LIN {X 0.035,Y -624.927,Z 1269.319,A 0.000,B 0.000,C 90.000,E1 93.326} C_DIS
LIN {X 0.207,Y -616.621,Z 1269.315,A 0.000,B 0.000,C 90.000,E1 92.636} C_DIS
LIN {X -0.076,Y -609.408,Z 1269.312,A 0.000,B 0.000,C 90.000,E1 92.121} C_DIS
LIN {X -0.106,Y -601.874,Z 1269.309,A 0.000,B 0.000,C 90.000,E1 91.604} C_DIS
LIN {X 0.134,Y -595.870,Z 1269.307,A 0.000,B 0.000,C 90.000,E1 91.203} C_DIS
LIN {X -0.159,Y -588.937,Z 1269.305,A 0.000,B 0.000,C 90.000,E1 90.859} C_DIS
LIN {X 0.273,Y -583.448,Z 1269.303,A 0.000,B 0.000,C 90.000,E1 90.573} C_DIS
LIN {X -0.248,Y -576.328,Z 1269.302,A 0.000,B 0.000,C 90.000,E1 90.344} C_DIS
LIN {X -0.083,Y -571.719,Z 1269.301,A 0.000,B 0.000,C 90.000,E1 90.115} C_DIS
LIN {X -0.130,Y -571.653,Z 1269.301,A 0.000,B 0.000,C 90.000,E1 90.115} C_DIS
LIN {X -0.005,Y -570.486,Z 1269.300,A 0.000,B 0.000,C 90.000,E1 89.943} C_DIS
LIN {X -0.259,Y -568.764,Z 1269.299,A 0.000,B 0.000,C 90.000,E1 89.771} C_DIS
LIN {X 0.268,Y -568.741,Z 1269.299,A 0.000,B 0.000,C 90.000,E1 89.714} C_DIS
LIN {X 0.075,Y -568.279,Z 1269.297,A 0.000,B 0.000,C 90.000,E1 89.370} C_DIS
LIN {X 0.099,Y -568.544,Z 1269.293,A 0.000,B 0.000,C 90.000,E1 88.682} C_DIS
LIN {X 0.005,Y -570.330,Z 1269.281,A 0.000,B 0.000,C 90.000,E1 86.502} C_DIS
LIN {X -0.257,Y -573.067,Z 1269.266,A 0.000,B 0.000,C 90.000,E1 83.799} C_DIS
LIN {X -0.006,Y -574.512,Z 1269.258,A 0.000,B 0.000,C 90.000,E1 82.413} C_DIS
LIN {X 0.063,Y -575.760,Z 1269.252,A 0.000,B 0.000,C 90.000,E1 81.319} C_DIS
LIN {X -0.129,Y -577.174,Z 1269.244,A 0.000,B 0.000,C 90.000,E1 79.982} C_DIS
LIN {X 0.162,Y -578.183,Z 1269.238,A 0.000,B 0.000,C 90.000,E1 78.870} C_DIS
LIN {X -0.213,Y -579.536,Z 1269.229,A 0.000,B 0.000,C 90.000,E1 77.285} C_DIS
LIN {X 0.115,Y -580.341,Z 1269.223,A 0.000,B 0.000,C 90.000,E1 76.172} C_DIS
LIN {X -0.086,Y -581.484,Z 1269.214,A 0.000,B 0.000,C 90.000,E1 74.574} C_DIS
LIN {X 0.110,Y -582.570,Z 1269.204,A 0.000,B 0.000,C 90.000,E1 72.670} C_DIS
LIN {X 0.220,Y -583.261,Z 1269.198,A 0.000,B 0.000,C 90.000,E1 71.583} C_DIS
LIN {X -0.147,Y -584.186,Z 1269.189,A 0.000,B 0.000,C 90.000,E1 70.007} C_DIS
LIN {X -0.142,Y -585.613,Z 1269.176,A 0.000,B 0.000,C 90.000,E1 67.592} C_DIS
LIN {X 0.272,Y -587.301,Z 1269.164,A 0.000,B 0.000,C 90.000,E1 65.409} C_DIS
LIN {X -0.020,Y -588.370,Z 1269.156,A 0.000,B 0.000,C 90.000,E1 64.101} C_DIS
LIN {X -0.109,Y -590.186,Z 1269.144,A 0.000,B 0.000,C 90.000,E1 61.975} C_DIS
LIN {X -0.172,Y -591.757,Z 1269.135,A 0.000,B 0.000,C 90.000,E1 60.383} C_DIS
LIN {X -0.394,Y -593.165,Z 1269.128,A 0.000,B 0.000,C 90.000,E1 59.076} C_DIS
LIN {X 0.019,Y -594.578,Z 1269.121,A 0.000,B 0.000,C 90.000,E1 57.709} C_DIS
LIN {X -0.137,Y -596.161,Z 1269.112,A 0.000,B 0.000,C 90.000,E1 56.135} C_DIS
LIN {X 0.075,Y -597.715,Z 1269.103,A 0.000,B 0.000,C 90.000,E1 54.529} C_DIS
LIN {X -0.172,Y -599.043,Z 1269.094,A 0.000,B 0.000,C 90.000,E1 52.970} C_DIS
LIN {X -0.032,Y -600.276,Z 1269.085,A 0.000,B 0.000,C 90.000,E1 51.376} C_DIS
LIN {X -0.367,Y -601.098,Z 1269.080,A 0.000,B 0.000,C 90.000,E1 50.356} C_DIS
LIN {X -0.097,Y -601.474,Z 1269.075,A 0.000,B 0.000,C 90.000,E1 49.542} C_DIS
LIN {X -0.018,Y -602.330,Z 1269.064,A 0.000,B 0.000,C 90.000,E1 47.433} C_DIS
LIN {X -0.156,Y -602.728,Z 1269.056,A 0.000,B 0.000,C 90.000,E1 46.134} C_DIS
LIN {X 0.091,Y -602.846,Z 1269.052,A 0.000,B 0.000,C 90.000,E1 45.324} C_DIS
LIN {X -0.063,Y -602.734,Z 1269.045,A 0.000,B 0.000,C 90.000,E1 44.028} C_DIS
LIN {X -0.024,Y -602.493,Z 1269.039,A 0.000,B 0.000,C 90.000,E1 42.975} C_DIS
LIN {X 0.077,Y -601.909,Z 1269.030,A 0.000,B 0.000,C 90.000,E1 41.391} C_DIS
LIN {X 0.179,Y -601.206,Z 1269.021,A 0.000,B 0.000,C 90.000,E1 39.806} C_DIS
LIN {X 0.231,Y -600.557,Z 1269.016,A 0.000,B 0.000,C 90.000,E1 38.749} C_DIS
LIN {X -0.104,Y -599.810,Z 1269.010,A 0.000,B 0.000,C 90.000,E1 37.729} C_DIS
LIN {X 0.267,Y -598.410,Z 1269.002,A 0.000,B 0.000,C 90.000,E1 36.377} C_DIS
LIN {X -0.218,Y -596.615,Z 1268.995,A 0.000,B 0.000,C 90.000,E1 35.105} C_DIS
LIN {X -0.248,Y -594.236,Z 1268.988,A 0.000,B 0.000,C 90.000,E1 33.785} C_DIS
LIN {X 0.075,Y -592.556,Z 1268.983,A 0.000,B 0.000,C 90.000,E1 32.959} C_DIS
LIN {X 0.173,Y -591.315,Z 1268.980,A 0.000,B 0.000,C 90.000,E1 32.418} C_DIS
LIN {X -0.160,Y -588.416,Z 1268.974,A 0.000,B 0.000,C 90.000,E1 31.386} C_DIS
LIN {X -0.215,Y -585.793,Z 1268.970,A 0.000,B 0.000,C 90.000,E1 30.590} C_DIS
LIN {X -0.167,Y -583.891,Z 1268.967,A 0.000,B 0.000,C 90.000,E1 30.050} C_DIS
LIN {X 0.238,Y -580.550,Z 1268.962,A 0.000,B 0.000,C 90.000,E1 29.205} C_DIS
LIN {X 0.026,Y -576.284,Z 1268.957,A 0.000,B 0.000,C 90.000,E1 28.281} C_DIS
LIN {X 0.075,Y -571.866,Z 1268.953,A 0.000,B 0.000,C 90.000,E1 27.462} C_DIS
LIN {X -0.166,Y -567.213,Z 1268.948,A 0.000,B 0.000,C 90.000,E1 26.668} C_DIS
LIN {X -0.204,Y -561.915,Z 1268.943,A 0.000,B 0.000,C 90.000,E1 25.848} C_DIS
LIN {X -0.191,Y -557.238,Z 1268.940,A 0.000,B 0.000,C 90.000,E1 25.155} C_DIS
LIN {X -0.002,Y -554.199,Z 1268.937,A 0.000,B 0.000,C 90.000,E1 24.719} C_DIS
LIN {X -0.172,Y -547.673,Z 1268.933,A 0.000,B 0.000,C 90.000,E1 23.898} C_DIS
LIN {X 0.087,Y -540.497,Z 1268.928,A 0.000,B 0.000,C 90.000,E1 23.025} C_DIS
LIN {X 0.186,Y -536.683,Z 1268.926,A 0.000,B 0.000,C 90.000,E1 22.589} C_DIS
LIN {X -0.022,Y -527.764,Z 1268.920,A 0.000,B 0.000,C 90.000,E1 21.642} C_DIS
LIN {X 0.012,Y -518.433,Z 1268.915,A 0.000,B 0.000,C 90.000,E1 20.663} C_DIS
LIN {X -0.089,Y -507.507,Z 1268.909,A 0.000,B 0.000,C 90.000,E1 19.577} C_DIS
LIN {X 0.166,Y -497.766,Z 1268.903,A 0.000,B 0.000,C 90.000,E1 18.598} C_DIS
LIN {X -0.088,Y -489.206,Z 1268.899,A 0.000,B 0.000,C 90.000,E1 17.819} C_DIS
LIN {X -0.222,Y -480.567,Z 1268.895,A 0.000,B 0.000,C 90.000,E1 17.040} C_DIS
LIN {X -0.066,Y -467.187,Z 1268.888,A 0.000,B 0.000,C 90.000,E1 15.843} C_DIS
LIN {X 0.059,Y -446.488,Z 1268.878,A 0.000,B 0.000,C 90.000,E1 13.939} C_DIS
LIN {X -0.007,Y -429.004,Z 1268.868,A 0.000,B 0.000,C 90.000,E1 12.243} C_DIS
LIN {X -0.023,Y -411.922,Z 1268.858,A 0.000,B 0.000,C 90.000,E1 10.433} C_DIS
LIN {X 0.080,Y -402.151,Z 1268.852,A 0.000,B 0.000,C 90.000,E1 9.321} C_DIS
LIN {X -0.078,Y -398.253,Z 1268.849,A 0.000,B 0.000,C 90.000,E1 8.859} C_DIS
LIN {X 0.174,Y -395.068,Z 1268.847,A 0.000,B 0.000,C 90.000,E1 8.341} C_DIS
LIN {X 0.205,Y -394.907,Z 1268.846,A 0.000,B 0.000,C 90.000,E1 8.276} C_DIS
LIN {X 0.167,Y -394.904,Z 1268.846,A 0.000,B 0.000,C 90.000,E1 8.276} C_DIS
LIN {X -0.182,Y -395.576,Z 1268.845,A 0.000,B 0.000,C 90.000,E1 8.106} C_DIS
LIN {X -0.008,Y -396.125,Z 1268.844,A 0.000,B 0.000,C 90.000,E1 7.992} C_DIS
LIN {X 0.069,Y -399.536,Z 1268.843,A 0.000,B 0.000,C 90.000,E1 7.644} C_DIS
LIN {X -0.190,Y -401.491,Z 1268.842,A 0.000,B 0.000,C 90.000,E1 7.530} C_DIS
LIN {X -0.044,Y -408.684,Z 1268.839,A 0.000,B 0.000,C 90.000,E1 7.068} C_DIS
LIN {X -0.067,Y -413.477,Z 1268.838,A 0.000,B 0.000,C 90.000,E1 6.777} C_DIS
LIN {X 0.129,Y -419.785,Z 1268.835,A 0.000,B 0.000,C 90.000,E1 6.315} C_DIS
LIN {X 0.092,Y -426.124,Z 1268.833,A 0.000,B 0.000,C 90.000,E1 5.853} C_DIS
LIN {X 0.180,Y -435.617,Z 1268.828,A 0.000,B 0.000,C 90.000,E1 5.106} C_DIS
LIN {X -0.122,Y -443.387,Z 1268.825,A 0.000,B 0.000,C 90.000,E1 4.531} C_DIS
LIN {X 0.118,Y -454.124,Z 1268.820,A 0.000,B 0.000,C 90.000,E1 3.612} C_DIS
LIN {X -0.027,Y -461.487,Z 1268.817,A 0.000,B 0.000,C 90.000,E1 2.980} C_DIS
LIN {X -0.200,Y -467.315,Z 1268.814,A 0.000,B 0.000,C 90.000,E1 2.465} C_DIS
LIN {X 0.179,Y -474.204,Z 1268.810,A 0.000,B 0.000,C 90.000,E1 1.718} C_DIS
LIN {X 0.163,Y -479.557,Z 1268.807,A 0.000,B 0.000,C 90.000,E1 1.146} C_DIS
LIN {X -0.200,Y -487.318,Z 1268.802,A 0.000,B 0.000,C 90.000,E1 0.286} C_DIS
LIN {X 0.026,Y -493.312,Z 1268.797,A 0.000,B 0.000,C 90.000,E1 359.484} C_DIS
LIN {X -0.091,Y -498.725,Z 1268.793,A 0.000,B 0.000,C 90.000,E1 358.740} C_DIS
LIN {X 0.049,Y -504.636,Z 1268.788,A 0.000,B 0.000,C 90.000,E1 357.822} C_DIS
LIN {X -0.171,Y -508.377,Z 1268.785,A 0.000,B 0.000,C 90.000,E1 357.249} C_DIS
LIN {X -0.132,Y -512.702,Z 1268.781,A 0.000,B 0.000,C 90.000,E1 356.502} C_DIS
LIN {X 0.249,Y -516.047,Z 1268.777,A 0.000,B 0.000,C 90.000,E1 355.869} C_DIS
LIN {X -0.149,Y -519.875,Z 1268.773,A 0.000,B 0.000,C 90.000,E1 355.179} C_DIS
LIN {X 0.003,Y -523.393,Z 1268.769,A 0.000,B 0.000,C 90.000,E1 354.432} C_DIS
LIN {X 0.199,Y -527.979,Z 1268.763,A 0.000,B 0.000,C 90.000,E1 353.394} C_DIS
LIN {X -0.078,Y -531.971,Z 1268.758,A 0.000,B 0.000,C 90.000,E1 352.413} C_DIS
LIN {X -0.036,Y -535.135,Z 1268.753,A 0.000,B 0.000,C 90.000,E1 351.546} C_DIS
LIN {X 0.039,Y -537.984,Z 1268.748,A 0.000,B 0.000,C 90.000,E1 350.679} C_DIS
LIN {X 0.233,Y -540.592,Z 1268.744,A 0.000,B 0.000,C 90.000,E1 349.803} C_DIS
LIN {X -0.094,Y -543.724,Z 1268.737,A 0.000,B 0.000,C 90.000,E1 348.701} C_DIS
LIN {X 0.075,Y -545.161,Z 1268.734,A 0.000,B 0.000,C 90.000,E1 348.117} C_DIS
LIN {X 0.130,Y -548.295,Z 1268.726,A 0.000,B 0.000,C 90.000,E1 346.700} C_DIS
LIN {X -0.098,Y -549.960,Z 1268.722,A 0.000,B 0.000,C 90.000,E1 345.880} C_DIS
LIN {X -0.067,Y -551.925,Z 1268.715,A 0.000,B 0.000,C 90.000,E1 344.755} C_DIS
LIN {X 0.144,Y -553.533,Z 1268.709,A 0.000,B 0.000,C 90.000,E1 343.614} C_DIS
LIN {X 0.110,Y -554.552,Z 1268.704,A 0.000,B 0.000,C 90.000,E1 342.779} C_DIS
LIN {X -0.164,Y -555.602,Z 1268.698,A 0.000,B 0.000,C 90.000,E1 341.692} C_DIS
LIN {X -0.187,Y -556.065,Z 1268.694,A 0.000,B 0.000,C 90.000,E1 340.859} C_DIS
LIN {X -0.131,Y -556.226,Z 1268.691,A 0.000,B 0.000,C 90.000,E1 340.296} C_DIS
LIN {X 0.035,Y -556.128,Z 1268.686,A 0.000,B 0.000,C 90.000,E1 339.444} C_DIS
LIN {X 0.195,Y -555.751,Z 1268.681,A 0.000,B 0.000,C 90.000,E1 338.592} C_DIS
LIN {X 0.119,Y -554.781,Z 1268.675,A 0.000,B 0.000,C 90.000,E1 337.486} C_DIS
LIN {X -0.042,Y -553.574,Z 1268.670,A 0.000,B 0.000,C 90.000,E1 336.666} C_DIS
LIN {X 0.294,Y -552.191,Z 1268.666,A 0.000,B 0.000,C 90.000,E1 335.793} C_DIS
LIN {X 0.144,Y -549.562,Z 1268.658,A 0.000,B 0.000,C 90.000,E1 334.409} C_DIS
LIN {X 0.167,Y -547.974,Z 1268.655,A 0.000,B 0.000,C 90.000,E1 333.845} C_DIS
LIN {X -0.072,Y -547.336,Z 1268.653,A 0.000,B 0.000,C 90.000,E1 333.589} C_DIS
LIN {X -0.066,Y -544.751,Z 1268.649,A 0.000,B 0.000,C 90.000,E1 332.743} C_DIS
LIN {X 0.170,Y -542.787,Z 1268.645,A 0.000,B 0.000,C 90.000,E1 332.153} C_DIS
LIN {X 0.000,Y -538.988,Z 1268.640,A 0.000,B 0.000,C 90.000,E1 331.179} C_DIS
LIN {X -0.086,Y -534.890,Z 1268.635,A 0.000,B 0.000,C 90.000,E1 330.333} C_DIS
LIN {X -0.074,Y -530.995,Z 1268.631,A 0.000,B 0.000,C 90.000,E1 329.616} C_DIS
LIN {X 0.169,Y -526.763,Z 1268.627,A 0.000,B 0.000,C 90.000,E1 328.869} C_DIS
LIN {X -0.179,Y -517.818,Z 1268.619,A 0.000,B 0.000,C 90.000,E1 327.454} C_DIS
LIN {X -0.054,Y -513.311,Z 1268.615,A 0.000,B 0.000,C 90.000,E1 326.707} C_DIS
LIN {X 0.052,Y -508.342,Z 1268.610,A 0.000,B 0.000,C 90.000,E1 325.722} C_DIS
LIN {X -0.041,Y -506.934,Z 1268.608,A 0.000,B 0.000,C 90.000,E1 325.435} C_DIS
LIN {X -0.019,Y -504.396,Z 1268.604,A 0.000,B 0.000,C 90.000,E1 324.689} C_DIS
LIN {X 0.177,Y -502.941,Z 1268.601,A 0.000,B 0.000,C 90.000,E1 324.069} C_DIS
LIN {X -0.048,Y -501.800,Z 1268.597,A 0.000,B 0.000,C 90.000,E1 323.497} C_DIS
LIN {X -0.094,Y -500.755,Z 1268.592,A 0.000,B 0.000,C 90.000,E1 322.603} C_DIS
LIN {X 0.129,Y -500.263,Z 1268.586,A 0.000,B 0.000,C 90.000,E1 321.376} C_DIS
LIN {X -0.162,Y -500.472,Z 1268.569,A 0.000,B 0.000,C 90.000,E1 318.405} C_DIS
LIN {X -0.183,Y -500.796,Z 1268.561,A 0.000,B 0.000,C 90.000,E1 316.905} C_DIS
LIN {X 0.016,Y -501.097,Z 1268.551,A 0.000,B 0.000,C 90.000,E1 315.081} C_DIS
LIN {X 0.012,Y -501.418,Z 1268.542,A 0.000,B 0.000,C 90.000,E1 313.581} C_DIS
LIN {X 0.098,Y -501.843,Z 1268.531,A 0.000,B 0.000,C 90.000,E1 311.472} C_DIS
LIN {X -0.319,Y -502.018,Z 1268.526,A 0.000,B 0.000,C 90.000,E1 310.620} C_DIS
LIN {X 0.198,Y -502.277,Z 1268.514,A 0.000,B 0.000,C 90.000,E1 308.463} C_DIS
LIN {X 0.215,Y -502.635,Z 1268.504,A 0.000,B 0.000,C 90.000,E1 306.664} C_DIS
LIN {X -0.241,Y -502.814,Z 1268.497,A 0.000,B 0.000,C 90.000,E1 305.518} C_DIS
LIN {X 0.012,Y -502.898,Z 1268.489,A 0.000,B 0.000,C 90.000,E1 303.992} C_DIS
LIN {X -0.008,Y -502.787,Z 1268.481,A 0.000,B 0.000,C 90.000,E1 302.498} C_DIS
LIN {X -0.336,Y -502.678,Z 1268.474,A 0.000,B 0.000,C 90.000,E1 301.337} C_DIS
LIN {X -0.020,Y -502.393,Z 1268.462,A 0.000,B 0.000,C 90.000,E1 299.205} C_DIS
LIN {X -0.041,Y -502.118,Z 1268.457,A 0.000,B 0.000,C 90.000,E1 298.309} C_DIS
LIN {X 0.174,Y -501.594,Z 1268.452,A 0.000,B 0.000,C 90.000,E1 297.385} C_DIS
LIN {X -0.236,Y -500.511,Z 1268.446,A 0.000,B 0.000,C 90.000,E1 296.232} C_DIS
LIN {X 0.112,Y -499.828,Z 1268.442,A 0.000,B 0.000,C 90.000,E1 295.591} C_DIS
LIN {X -0.210,Y -498.815,Z 1268.439,A 0.000,B 0.000,C 90.000,E1 295.027} C_DIS
LIN {X -0.146,Y -498.129,Z 1268.437,A 0.000,B 0.000,C 90.000,E1 294.719} C_DIS
LIN {X 0.123,Y -497.166,Z 1268.436,A 0.000,B 0.000,C 90.000,E1 294.387} C_DIS
LIN {X 0.115,Y -484.996,Z 1268.417,A 0.000,B 0.000,C 90.000,E1 291.046} C_DIS
LIN {X 0.200,Y -474.861,Z 1268.398,A 0.000,B 0.000,C 90.000,E1 287.638} C_DIS
LIN {X 0.148,Y -466.026,Z 1268.377,A 0.000,B 0.000,C 90.000,E1 283.883} C_DIS
LIN {X 0.122,Y -458.541,Z 1268.353,A 0.000,B 0.000,C 90.000,E1 279.443} C_DIS
LIN {X -0.148,Y -453.086,Z 1268.319,A 0.000,B 0.000,C 90.000,E1 273.383} C_DIS
LIN {X -0.186,Y -456.218,Z 1268.260,A 0.000,B 0.000,C 90.000,E1 262.761} C_DIS
LIN {X 0.082,Y -462.985,Z 1268.233,A 0.000,B 0.000,C 90.000,E1 257.937} C_DIS
LIN {X -0.066,Y -471.652,Z 1268.210,A 0.000,B 0.000,C 90.000,E1 253.850} C_DIS
LIN {X 0.201,Y -472.429,Z 1268.208,A 0.000,B 0.000,C 90.000,E1 253.504} C_DIS
LIN {X 0.154,Y -473.058,Z 1268.207,A 0.000,B 0.000,C 90.000,E1 253.196} C_DIS
LIN {X -0.070,Y -473.773,Z 1268.203,A 0.000,B 0.000,C 90.000,E1 252.598} C_DIS
LIN {X 0.127,Y -474.288,Z 1268.198,A 0.000,B 0.000,C 90.000,E1 251.638} C_DIS
LIN {X -0.122,Y -474.509,Z 1268.193,A 0.000,B 0.000,C 90.000,E1 250.732} C_DIS
LIN {X 0.238,Y -474.453,Z 1268.188,A 0.000,B 0.000,C 90.000,E1 249.752} C_DIS
LIN {X -0.076,Y -474.004,Z 1268.179,A 0.000,B 0.000,C 90.000,E1 248.230} C_DIS
LIN {X -0.136,Y -473.655,Z 1268.176,A 0.000,B 0.000,C 90.000,E1 247.614} C_DIS
LIN {X -0.150,Y -472.547,Z 1268.165,A 0.000,B 0.000,C 90.000,E1 245.741} C_DIS
LIN {X 0.048,Y -471.538,Z 1268.156,A 0.000,B 0.000,C 90.000,E1 244.152} C_DIS
LIN {X -0.087,Y -470.205,Z 1268.144,A 0.000,B 0.000,C 90.000,E1 241.975} C_DIS
LIN {X 0.091,Y -469.264,Z 1268.136,A 0.000,B 0.000,C 90.000,E1 240.383} C_DIS
LIN {X 0.099,Y -468.521,Z 1268.129,A 0.000,B 0.000,C 90.000,E1 239.125} C_DIS
LIN {X -0.153,Y -467.371,Z 1268.120,A 0.000,B 0.000,C 90.000,E1 237.582} C_DIS
LIN {X -0.130,Y -465.545,Z 1268.106,A 0.000,B 0.000,C 90.000,E1 235.055} C_DIS
LIN {X 0.093,Y -464.433,Z 1268.095,A 0.000,B 0.000,C 90.000,E1 233.130} C_DIS
LIN {X 0.121,Y -463.067,Z 1268.079,A 0.000,B 0.000,C 90.000,E1 230.275} C_DIS
LIN {X -0.149,Y -462.397,Z 1268.069,A 0.000,B 0.000,C 90.000,E1 228.405} C_DIS
LIN {X 0.126,Y -461.835,Z 1268.060,A 0.000,B 0.000,C 90.000,E1 226.782} C_DIS
LIN {X -0.229,Y -461.215,Z 1268.049,A 0.000,B 0.000,C 90.000,E1 224.919} C_DIS
LIN {X -0.069,Y -460.783,Z 1268.021,A 0.000,B 0.000,C 90.000,E1 219.806} C_DIS
LIN {X -0.138,Y -461.727,Z 1268.005,A 0.000,B 0.000,C 90.000,E1 216.950} C_DIS
LIN {X -0.167,Y -465.801,Z 1267.977,A 0.000,B 0.000,C 90.000,E1 211.878} C_DIS
LIN {X -0.070,Y -469.126,Z 1267.961,A 0.000,B 0.000,C 90.000,E1 209.027} C_DIS
LIN {X -0.124,Y -470.925,Z 1267.953,A 0.000,B 0.000,C 90.000,E1 207.462} C_DIS
LIN {X -0.109,Y -474.555,Z 1267.937,A 0.000,B 0.000,C 90.000,E1 204.643} C_DIS
LIN {X -0.076,Y -477.435,Z 1267.927,A 0.000,B 0.000,C 90.000,E1 202.770} C_DIS
LIN {X 0.272,Y -482.630,Z 1267.909,A 0.000,B 0.000,C 90.000,E1 199.631} C_DIS
LIN {X -0.030,Y -485.453,Z 1267.901,A 0.000,B 0.000,C 90.000,E1 198.127} C_DIS
LIN {X 0.079,Y -489.644,Z 1267.889,A 0.000,B 0.000,C 90.000,E1 195.969} C_DIS
LIN {X 0.060,Y -494.390,Z 1267.875,A 0.000,B 0.000,C 90.000,E1 193.536} C_DIS
LIN {X 0.109,Y -498.139,Z 1267.865,A 0.000,B 0.000,C 90.000,E1 191.715} C_DIS
LIN {X 0.142,Y -501.925,Z 1267.855,A 0.000,B 0.000,C 90.000,E1 189.905} C_DIS
LIN {X 0.170,Y -505.704,Z 1267.845,A 0.000,B 0.000,C 90.000,E1 188.106} C_DIS
LIN {X -0.243,Y -508.929,Z 1267.837,A 0.000,B 0.000,C 90.000,E1 186.663} C_DIS
LIN {X -0.094,Y -512.117,Z 1267.829,A 0.000,B 0.000,C 90.000,E1 185.163} C_DIS
LIN {X -0.011,Y -515.813,Z 1267.819,A 0.000,B 0.000,C 90.000,E1 183.383} C_DIS
LIN {X 0.151,Y -519.393,Z 1267.809,A 0.000,B 0.000,C 90.000,E1 181.604} C_DIS
LIN {X -0.164,Y -522.786,Z 1267.799,A 0.000,B 0.000,C 90.000,E1 179.885} C_DIS
LIN {X 0.153,Y -525.585,Z 1267.791,A 0.000,B 0.000,C 90.000,E1 178.396} C_DIS
LIN {X 0.036,Y -527.664,Z 1267.785,A 0.000,B 0.000,C 90.000,E1 177.249} C_DIS
LIN {X -0.051,Y -529.596,Z 1267.778,A 0.000,B 0.000,C 90.000,E1 176.102} C_DIS
LIN {X -0.096,Y -531.738,Z 1267.770,A 0.000,B 0.000,C 90.000,E1 174.666} C_DIS
LIN {X -0.062,Y -532.903,Z 1267.766,A 0.000,B 0.000,C 90.000,E1 173.799} C_DIS
LIN {X -0.034,Y -534.234,Z 1267.759,A 0.000,B 0.000,C 90.000,E1 172.648} C_DIS
LIN {X 0.081,Y -535.419,Z 1267.753,A 0.000,B 0.000,C 90.000,E1 171.489} C_DIS
LIN {X 0.157,Y -536.247,Z 1267.748,A 0.000,B 0.000,C 90.000,E1 170.622} C_DIS
LIN {X -0.258,Y -536.720,Z 1267.745,A 0.000,B 0.000,C 90.000,E1 170.095} C_DIS
LIN {X -0.012,Y -537.474,Z 1267.739,A 0.000,B 0.000,C 90.000,E1 168.926} C_DIS
LIN {X 0.247,Y -538.044,Z 1267.732,A 0.000,B 0.000,C 90.000,E1 167.757} C_DIS
LIN {X -0.017,Y -538.443,Z 1267.726,A 0.000,B 0.000,C 90.000,E1 166.645} C_DIS
LIN {X -0.087,Y -538.864,Z 1267.718,A 0.000,B 0.000,C 90.000,E1 165.227} C_DIS
LIN {X 0.137,Y -540.453,Z 1267.701,A 0.000,B 0.000,C 90.000,E1 162.072} C_DIS
LIN {X -0.109,Y -542.157,Z 1267.693,A 0.000,B 0.000,C 90.000,E1 160.678} C_DIS
LIN {X 0.137,Y -544.217,Z 1267.686,A 0.000,B 0.000,C 90.000,E1 159.518} C_DIS
LIN {X 0.164,Y -546.283,Z 1267.682,A 0.000,B 0.000,C 90.000,E1 158.666} C_DIS
LIN {X -0.094,Y -548.817,Z 1267.677,A 0.000,B 0.000,C 90.000,E1 157.847} C_DIS
LIN {X 0.130,Y -553.710,Z 1267.670,A 0.000,B 0.000,C 90.000,E1 156.561} C_DIS
LIN {X -0.325,Y -556.414,Z 1267.667,A 0.000,B 0.000,C 90.000,E1 156.049} C_DIS
LIN {X -0.156,Y -562.817,Z 1267.661,A 0.000,B 0.000,C 90.000,E1 154.921} C_DIS
LIN {X -0.158,Y -569.964,Z 1267.655,A 0.000,B 0.000,C 90.000,E1 153.819} C_DIS
LIN {X -0.230,Y -576.497,Z 1267.649,A 0.000,B 0.000,C 90.000,E1 152.871} C_DIS
LIN {X 0.111,Y -582.405,Z 1267.645,A 0.000,B 0.000,C 90.000,E1 152.025} C_DIS
LIN {X -0.138,Y -587.280,Z 1267.641,A 0.000,B 0.000,C 90.000,E1 151.385} C_DIS
LIN {X -0.143,Y -591.984,Z 1267.637,A 0.000,B 0.000,C 90.000,E1 150.717} C_DIS
LIN {X -0.351,Y -595.788,Z 1267.634,A 0.000,B 0.000,C 90.000,E1 150.205} C_DIS
LIN {X -0.185,Y -601.127,Z 1267.630,A 0.000,B 0.000,C 90.000,E1 149.410} C_DIS
LIN {X -0.003,Y -607.111,Z 1267.625,A 0.000,B 0.000,C 90.000,E1 148.486} C_DIS
LIN {X 0.136,Y -613.688,Z 1267.619,A 0.000,B 0.000,C 90.000,E1 147.454} C_DIS
LIN {X 0.119,Y -620.570,Z 1267.613,A 0.000,B 0.000,C 90.000,E1 146.294} C_DIS
LIN {X -0.115,Y -624.053,Z 1267.609,A 0.000,B 0.000,C 90.000,E1 145.674} C_DIS
LIN {X 0.021,Y -628.643,Z 1267.604,A 0.000,B 0.000,C 90.000,E1 144.769} C_DIS
LIN {X 0.213,Y -632.293,Z 1267.600,A 0.000,B 0.000,C 90.000,E1 143.989} C_DIS
LIN {X 0.066,Y -634.590,Z 1267.597,A 0.000,B 0.000,C 90.000,E1 143.497} C_DIS
LIN {X -0.196,Y -637.668,Z 1267.593,A 0.000,B 0.000,C 90.000,E1 142.763} C_DIS
LIN {X -0.024,Y -641.477,Z 1267.588,A 0.000,B 0.000,C 90.000,E1 141.743} C_DIS
LIN {X -0.120,Y -643.313,Z 1267.585,A 0.000,B 0.000,C 90.000,E1 141.251} C_DIS
LIN {X 0.042,Y -647.393,Z 1267.578,A 0.000,B 0.000,C 90.000,E1 139.989} C_DIS
LIN {X -0.097,Y -649.646,Z 1267.574,A 0.000,B 0.000,C 90.000,E1 139.256} C_DIS
LIN {X 0.104,Y -653.340,Z 1267.567,A 0.000,B 0.000,C 90.000,E1 138.000} C_DIS
LIN {X -0.032,Y -656.183,Z 1267.561,A 0.000,B 0.000,C 90.000,E1 137.025} C_DIS
LIN {X -0.291,Y -663.170,Z 1267.548,A 0.000,B 0.000,C 90.000,E1 134.595} C_DIS
LIN {X 0.148,Y -667.555,Z 1267.540,A 0.000,B 0.000,C 90.000,E1 133.095} C_DIS
LIN {X -0.283,Y -671.215,Z 1267.533,A 0.000,B 0.000,C 90.000,E1 131.919} C_DIS
LIN {X -0.143,Y -675.448,Z 1267.525,A 0.000,B 0.000,C 90.000,E1 130.458} C_DIS
LIN {X -0.390,Y -678.875,Z 1267.518,A 0.000,B 0.000,C 90.000,E1 129.277} C_DIS
LIN {X -0.017,Y -682.789,Z 1267.510,A 0.000,B 0.000,C 90.000,E1 127.810} C_DIS
LIN {X 0.392,Y -685.906,Z 1267.503,A 0.000,B 0.000,C 90.000,E1 126.583} C_DIS
LIN {X 0.079,Y -689.362,Z 1267.496,A 0.000,B 0.000,C 90.000,E1 125.185} C_DIS
LIN {X -0.023,Y -691.528,Z 1267.490,A 0.000,B 0.000,C 90.000,E1 124.246} C_DIS
LIN {X -0.275,Y -693.944,Z 1267.484,A 0.000,B 0.000,C 90.000,E1 123.086} C_DIS
LIN {X 0.102,Y -696.275,Z 1267.477,A 0.000,B 0.000,C 90.000,E1 121.878} C_DIS
LIN {X -0.078,Y -698.431,Z 1267.471,A 0.000,B 0.000,C 90.000,E1 120.718} C_DIS
LIN {X 0.016,Y -700.220,Z 1267.464,A 0.000,B 0.000,C 90.000,E1 119.539} C_DIS
LIN {X -0.131,Y -701.512,Z 1267.459,A 0.000,B 0.000,C 90.000,E1 118.615} C_DIS
LIN {X 0.075,Y -702.377,Z 1267.455,A 0.000,B 0.000,C 90.000,E1 117.897} C_DIS
LIN {X -0.377,Y -703.226,Z 1267.450,A 0.000,B 0.000,C 90.000,E1 117.001} C_DIS
LIN {X -0.160,Y -703.486,Z 1267.446,A 0.000,B 0.000,C 90.000,E1 116.283} C_DIS
LIN {X 0.098,Y -703.536,Z 1267.443,A 0.000,B 0.000,C 90.000,E1 115.796} C_DIS
LIN {X 0.313,Y -703.254,Z 1267.440,A 0.000,B 0.000,C 90.000,E1 115.079} C_DIS
LIN {X -0.059,Y -702.876,Z 1267.437,A 0.000,B 0.000,C 90.000,E1 114.643} C_DIS
LIN {X 0.212,Y -702.100,Z 1267.434,A 0.000,B 0.000,C 90.000,E1 114.155} C_DIS
LIN {X -0.152,Y -701.468,Z 1267.433,A 0.000,B 0.000,C 90.000,E1 113.951} C_DIS
LIN {X 0.113,Y -699.633,Z 1267.430,A 0.000,B 0.000,C 90.000,E1 113.462} C_DIS
LIN {X 0.248,Y -698.955,Z 1267.430,A 0.000,B 0.000,C 90.000,E1 113.334} C_DIS
LIN {X -0.094,Y -694.975,Z 1267.427,A 0.000,B 0.000,C 90.000,E1 112.898} C_DIS
LIN {X 0.083,Y -693.840,Z 1267.427,A 0.000,B 0.000,C 90.000,E1 112.770} C_DIS
LIN {X 0.210,Y -692.033,Z 1267.426,A 0.000,B 0.000,C 90.000,E1 112.642} C_DIS
LIN {X 0.122,Y -687.548,Z 1267.425,A 0.000,B 0.000,C 90.000,E1 112.461} C_DIS
LIN {X 0.172,Y -684.871,Z 1267.424,A 0.000,B 0.000,C 90.000,E1 112.386} C_DIS
LIN {X -0.303,Y -681.996,Z 1267.424,A 0.000,B 0.000,C 90.000,E1 112.333} C_DIS
LIN {X -0.284,Y -679.939,Z 1267.424,A 0.000,B 0.000,C 90.000,E1 112.280} C_DIS
LIN {X -0.007,Y -676.149,Z 1267.423,A 0.000,B 0.000,C 90.000,E1 112.206} C_DIS
LIN {X 0.160,Y -670.243,Z 1267.423,A 0.000,B 0.000,C 90.000,E1 112.153} C_DIS
LIN {X 0.088,Y -634.230,Z 1267.423,A 0.000,B 0.000,C 90.000,E1 112.153} C_DIS
LIN {X 0.103,Y -632.331,Z 1267.423,A 0.000,B 0.000,C 90.000,E1 112.099} C_DIS
LIN {X -0.041,Y -631.528,Z 1267.423,A 0.000,B 0.000,C 90.000,E1 112.078} C_DIS
LIN {X -0.104,Y -631.458,Z 1267.423,A 0.000,B 0.000,C 90.000,E1 112.078} C_DIS
LIN {X 0.086,Y -631.183,Z 1267.422,A 0.000,B 0.000,C 90.000,E1 112.025} C_DIS
LIN {X 0.039,Y -631.152,Z 1267.422,A 0.000,B 0.000,C 90.000,E1 112.025} C_DIS
LIN {X -0.050,Y -631.304,Z 1267.421,A 0.000,B 0.000,C 90.000,E1 111.844} C_DIS
LIN {X 0.016,Y -634.446,Z 1267.418,A 0.000,B 0.000,C 90.000,E1 111.280} C_DIS
LIN {X -0.321,Y -640.403,Z 1267.413,A 0.000,B 0.000,C 90.000,E1 110.429} C_DIS
LIN {X 0.153,Y -643.671,Z 1267.411,A 0.000,B 0.000,C 90.000,E1 109.885} C_DIS
LIN {X 0.105,Y -647.861,Z 1267.406,A 0.000,B 0.000,C 90.000,E1 109.141} C_DIS
LIN {X -0.089,Y -652.257,Z 1267.402,A 0.000,B 0.000,C 90.000,E1 108.290} C_DIS
LIN {X 0.222,Y -656.902,Z 1267.396,A 0.000,B 0.000,C 90.000,E1 107.275} C_DIS
LIN {X 0.073,Y -660.098,Z 1267.392,A 0.000,B 0.000,C 90.000,E1 106.551} C_DIS
LIN {X -0.233,Y -662.904,Z 1267.388,A 0.000,B 0.000,C 90.000,E1 105.843} C_DIS
LIN {X 0.308,Y -665.289,Z 1267.384,A 0.000,B 0.000,C 90.000,E1 105.064} C_DIS
LIN {X 0.138,Y -666.618,Z 1267.381,A 0.000,B 0.000,C 90.000,E1 104.592} C_DIS
LIN {X -0.101,Y -668.135,Z 1267.377,A 0.000,B 0.000,C 90.000,E1 103.883} C_DIS
LIN {X -0.253,Y -668.904,Z 1267.374,A 0.000,B 0.000,C 90.000,E1 103.411} C_DIS
LIN {X 0.181,Y -669.617,Z 1267.370,A 0.000,B 0.000,C 90.000,E1 102.647} C_DIS
LIN {X -0.104,Y -669.856,Z 1267.368,A 0.000,B 0.000,C 90.000,E1 102.187} C_DIS
LIN {X -0.244,Y -669.812,Z 1267.365,A 0.000,B 0.000,C 90.000,E1 101.715} C_DIS
LIN {X 0.197,Y -669.309,Z 1267.361,A 0.000,B 0.000,C 90.000,E1 100.950} C_DIS
LIN {X -0.153,Y -668.298,Z 1267.357,A 0.000,B 0.000,C 90.000,E1 100.254} C_DIS
LIN {X -0.232,Y -667.918,Z 1267.356,A 0.000,B 0.000,C 90.000,E1 100.018} C_DIS
LIN {X 0.150,Y -666.791,Z 1267.353,A 0.000,B 0.000,C 90.000,E1 99.500} C_DIS
LIN {X -0.024,Y -665.341,Z 1267.350,A 0.000,B 0.000,C 90.000,E1 99.029} C_DIS
LIN {X -0.218,Y -664.542,Z 1267.349,A 0.000,B 0.000,C 90.000,E1 98.803} C_DIS
LIN {X 0.245,Y -662.568,Z 1267.346,A 0.000,B 0.000,C 90.000,E1 98.276} C_DIS
LIN {X -0.160,Y -659.674,Z 1267.343,A 0.000,B 0.000,C 90.000,E1 97.701} C_DIS
LIN {X 0.172,Y -657.030,Z 1267.340,A 0.000,B 0.000,C 90.000,E1 97.182} C_DIS
LIN {X -0.270,Y -653.182,Z 1267.337,A 0.000,B 0.000,C 90.000,E1 96.606} C_DIS
LIN {X -0.025,Y -648.728,Z 1267.333,A 0.000,B 0.000,C 90.000,E1 95.967} C_DIS
LIN {X 0.167,Y -644.843,Z 1267.330,A 0.000,B 0.000,C 90.000,E1 95.454} C_DIS
LIN {X -0.245,Y -640.488,Z 1267.328,A 0.000,B 0.000,C 90.000,E1 94.992} C_DIS
LIN {X -0.047,Y -635.750,Z 1267.325,A 0.000,B 0.000,C 90.000,E1 94.473} C_DIS
LIN {X 0.211,Y -629.523,Z 1267.322,A 0.000,B 0.000,C 90.000,E1 93.841} C_DIS
LIN {X -0.010,Y -624.230,Z 1267.319,A 0.000,B 0.000,C 90.000,E1 93.383} C_DIS
LIN {X 0.075,Y -615.754,Z 1267.315,A 0.000,B 0.000,C 90.000,E1 92.694} C_DIS
LIN {X -0.226,Y -608.409,Z 1267.312,A 0.000,B 0.000,C 90.000,E1 92.178} C_DIS
LIN {X -0.262,Y -600.826,Z 1267.309,A 0.000,B 0.000,C 90.000,E1 91.661} C_DIS
LIN {X 0.255,Y -596.238,Z 1267.307,A 0.000,B 0.000,C 90.000,E1 91.318} C_DIS
LIN {X 0.138,Y -589.704,Z 1267.306,A 0.000,B 0.000,C 90.000,E1 90.974} C_DIS
LIN {X -0.174,Y -582.785,Z 1267.304,A 0.000,B 0.000,C 90.000,E1 90.688} C_DIS
LIN {X -0.083,Y -575.730,Z 1267.302,A 0.000,B 0.000,C 90.000,E1 90.401} C_DIS
LIN {X 0.208,Y -572.561,Z 1267.301,A 0.000,B 0.000,C 90.000,E1 90.229} C_DIS
LIN {X 0.028,Y -571.160,Z 1267.301,A 0.000,B 0.000,C 90.000,E1 90.172} C_DIS
LIN {X -0.151,Y -570.312,Z 1267.301,A 0.000,B 0.000,C 90.000,E1 90.115} C_DIS
LIN {X -0.255,Y -568.740,Z 1267.299,A 0.000,B 0.000,C 90.000,E1 89.885} C_DIS
LIN {X 0.272,Y -568.723,Z 1267.299,A 0.000,B 0.000,C 90.000,E1 89.828} C_DIS
LIN {X 0.066,Y -568.160,Z 1267.297,A 0.000,B 0.000,C 90.000,E1 89.370} C_DIS
LIN {X 0.212,Y -568.651,Z 1267.291,A 0.000,B 0.000,C 90.000,E1 88.396} C_DIS
LIN {X -0.006,Y -570.267,Z 1267.281,A 0.000,B 0.000,C 90.000,E1 86.502} C_DIS
LIN {X 0.116,Y -572.713,Z 1267.267,A 0.000,B 0.000,C 90.000,E1 84.033} C_DIS
LIN {X -0.216,Y -574.173,Z 1267.259,A 0.000,B 0.000,C 90.000,E1 82.704} C_DIS
LIN {X 0.252,Y -575.975,Z 1267.250,A 0.000,B 0.000,C 90.000,E1 81.027} C_DIS
LIN {X 0.066,Y -577.347,Z 1267.243,A 0.000,B 0.000,C 90.000,E1 79.690} C_DIS
LIN {X 0.144,Y -578.073,Z 1267.238,A 0.000,B 0.000,C 90.000,E1 78.870} C_DIS
LIN {X 0.331,Y -579.393,Z 1267.229,A 0.000,B 0.000,C 90.000,E1 77.229} C_DIS
LIN {X -0.249,Y -580.378,Z 1267.222,A 0.000,B 0.000,C 90.000,E1 75.936} C_DIS
LIN {X -0.112,Y -581.315,Z 1267.214,A 0.000,B 0.000,C 90.000,E1 74.574} C_DIS
LIN {X -0.138,Y -582.248,Z 1267.205,A 0.000,B 0.000,C 90.000,E1 72.960} C_DIS
LIN {X 0.188,Y -583.090,Z 1267.198,A 0.000,B 0.000,C 90.000,E1 71.583} C_DIS
LIN {X 0.159,Y -583.881,Z 1267.190,A 0.000,B 0.000,C 90.000,E1 70.242} C_DIS
LIN {X 0.076,Y -585.088,Z 1267.178,A 0.000,B 0.000,C 90.000,E1 68.103} C_DIS
LIN {X 0.227,Y -587.155,Z 1267.164,A 0.000,B 0.000,C 90.000,E1 65.409} C_DIS
LIN {X -0.068,Y -588.230,Z 1267.156,A 0.000,B 0.000,C 90.000,E1 64.101} C_DIS
LIN {X -0.160,Y -590.064,Z 1267.144,A 0.000,B 0.000,C 90.000,E1 61.975} C_DIS
LIN {X 0.288,Y -591.654,Z 1267.135,A 0.000,B 0.000,C 90.000,E1 60.333} C_DIS
LIN {X 0.363,Y -593.040,Z 1267.128,A 0.000,B 0.000,C 90.000,E1 58.997} C_DIS
LIN {X -0.040,Y -594.447,Z 1267.121,A 0.000,B 0.000,C 90.000,E1 57.709} C_DIS
LIN {X 0.297,Y -596.054,Z 1267.112,A 0.000,B 0.000,C 90.000,E1 56.087} C_DIS
LIN {X 0.011,Y -597.588,Z 1267.103,A 0.000,B 0.000,C 90.000,E1 54.529} C_DIS
LIN {X 0.240,Y -598.914,Z 1267.094,A 0.000,B 0.000,C 90.000,E1 52.924} C_DIS
LIN {X -0.101,Y -600.149,Z 1267.085,A 0.000,B 0.000,C 90.000,E1 51.376} C_DIS
LIN {X 0.024,Y -600.959,Z 1267.080,A 0.000,B 0.000,C 90.000,E1 50.312} C_DIS
LIN {X 0.071,Y -601.380,Z 1267.074,A 0.000,B 0.000,C 90.000,E1 49.256} C_DIS
LIN {X 0.111,Y -602.029,Z 1267.065,A 0.000,B 0.000,C 90.000,E1 47.676} C_DIS
LIN {X -0.062,Y -602.345,Z 1267.061,A 0.000,B 0.000,C 90.000,E1 46.905} C_DIS
LIN {X -0.006,Y -602.612,Z 1267.055,A 0.000,B 0.000,C 90.000,E1 45.850} C_DIS
LIN {X 0.031,Y -602.683,Z 1267.049,A 0.000,B 0.000,C 90.000,E1 44.798} C_DIS
LIN {X 0.299,Y -602.485,Z 1267.042,A 0.000,B 0.000,C 90.000,E1 43.461} C_DIS
LIN {X 0.160,Y -602.065,Z 1267.034,A 0.000,B 0.000,C 90.000,E1 42.162} C_DIS
LIN {X 0.022,Y -601.544,Z 1267.027,A 0.000,B 0.000,C 90.000,E1 40.862} C_DIS
LIN {X 0.086,Y -601.038,Z 1267.021,A 0.000,B 0.000,C 90.000,E1 39.806} C_DIS
LIN {X 0.137,Y -600.386,Z 1267.015,A 0.000,B 0.000,C 90.000,E1 38.749} C_DIS
LIN {X -0.201,Y -599.624,Z 1267.010,A 0.000,B 0.000,C 90.000,E1 37.729} C_DIS
LIN {X 0.169,Y -598.201,Z 1267.002,A 0.000,B 0.000,C 90.000,E1 36.377} C_DIS
LIN {X -0.321,Y -596.399,Z 1266.995,A 0.000,B 0.000,C 90.000,E1 35.105} C_DIS
LIN {X 0.250,Y -594.497,Z 1266.989,A 0.000,B 0.000,C 90.000,E1 33.992} C_DIS
LIN {X 0.079,Y -592.906,Z 1266.985,A 0.000,B 0.000,C 90.000,E1 33.214} C_DIS
LIN {X 0.064,Y -591.099,Z 1266.980,A 0.000,B 0.000,C 90.000,E1 32.418} C_DIS
LIN {X 0.230,Y -588.173,Z 1266.974,A 0.000,B 0.000,C 90.000,E1 31.337} C_DIS
LIN {X 0.176,Y -585.533,Z 1266.970,A 0.000,B 0.000,C 90.000,E1 30.541} C_DIS
LIN {X 0.224,Y -583.623,Z 1266.967,A 0.000,B 0.000,C 90.000,E1 30.001} C_DIS
LIN {X 0.120,Y -580.270,Z 1266.962,A 0.000,B 0.000,C 90.000,E1 29.205} C_DIS
LIN {X -0.023,Y -576.554,Z 1266.958,A 0.000,B 0.000,C 90.000,E1 28.409} C_DIS
LIN {X 0.260,Y -574.534,Z 1266.956,A 0.000,B 0.000,C 90.000,E1 27.975} C_DIS
LIN {X 0.047,Y -570.045,Z 1266.951,A 0.000,B 0.000,C 90.000,E1 27.180} C_DIS
LIN {X 0.124,Y -566.012,Z 1266.947,A 0.000,B 0.000,C 90.000,E1 26.488} C_DIS
LIN {X -0.025,Y -559.742,Z 1266.942,A 0.000,B 0.000,C 90.000,E1 25.540} C_DIS
LIN {X -0.029,Y -554.830,Z 1266.938,A 0.000,B 0.000,C 90.000,E1 24.847} C_DIS
LIN {X 0.147,Y -549.437,Z 1266.934,A 0.000,B 0.000,C 90.000,E1 24.131} C_DIS
LIN {X -0.170,Y -543.685,Z 1266.930,A 0.000,B 0.000,C 90.000,E1 23.462} C_DIS
LIN {X -0.272,Y -537.586,Z 1266.926,A 0.000,B 0.000,C 90.000,E1 22.770} C_DIS
LIN {X 0.089,Y -528.774,Z 1266.921,A 0.000,B 0.000,C 90.000,E1 21.770} C_DIS
LIN {X -0.014,Y -518.020,Z 1266.915,A 0.000,B 0.000,C 90.000,E1 20.663} C_DIS
LIN {X 0.012,Y -507.288,Z 1266.909,A 0.000,B 0.000,C 90.000,E1 19.577} C_DIS
LIN {X 0.047,Y -496.067,Z 1266.903,A 0.000,B 0.000,C 90.000,E1 18.489} C_DIS
LIN {X -0.235,Y -486.081,Z 1266.898,A 0.000,B 0.000,C 90.000,E1 17.583} C_DIS
LIN {X -0.218,Y -477.402,Z 1266.893,A 0.000,B 0.000,C 90.000,E1 16.804} C_DIS
LIN {X -0.011,Y -464.139,Z 1266.887,A 0.000,B 0.000,C 90.000,E1 15.607} C_DIS
LIN {X 0.164,Y -444.994,Z 1266.877,A 0.000,B 0.000,C 90.000,E1 13.828} C_DIS
LIN {X -0.118,Y -423.370,Z 1266.865,A 0.000,B 0.000,C 90.000,E1 11.715} C_DIS
LIN {X -0.068,Y -406.176,Z 1266.855,A 0.000,B 0.000,C 90.000,E1 9.849} C_DIS
LIN {X 0.178,Y -399.491,Z 1266.850,A 0.000,B 0.000,C 90.000,E1 9.029} C_DIS
LIN {X 0.195,Y -398.226,Z 1266.849,A 0.000,B 0.000,C 90.000,E1 8.859} C_DIS
LIN {X -0.213,Y -394.907,Z 1266.847,A 0.000,B 0.000,C 90.000,E1 8.398} C_DIS
LIN {X -0.087,Y -394.804,Z 1266.846,A 0.000,B 0.000,C 90.000,E1 8.341} C_DIS
LIN {X -0.125,Y -394.805,Z 1266.846,A 0.000,B 0.000,C 90.000,E1 8.341} C_DIS
LIN {X 0.187,Y -395.665,Z 1266.845,A 0.000,B 0.000,C 90.000,E1 8.049} C_DIS
LIN {X 0.139,Y -396.563,Z 1266.844,A 0.000,B 0.000,C 90.000,E1 7.936} C_DIS
LIN {X -0.070,Y -399.354,Z 1266.843,A 0.000,B 0.000,C 90.000,E1 7.701} C_DIS
LIN {X 0.112,Y -401.083,Z 1266.842,A 0.000,B 0.000,C 90.000,E1 7.530} C_DIS
LIN {X -0.006,Y -408.592,Z 1266.839,A 0.000,B 0.000,C 90.000,E1 7.068} C_DIS
LIN {X -0.021,Y -415.135,Z 1266.837,A 0.000,B 0.000,C 90.000,E1 6.663} C_DIS
LIN {X 0.106,Y -421.473,Z 1266.835,A 0.000,B 0.000,C 90.000,E1 6.201} C_DIS
LIN {X 0.032,Y -427.780,Z 1266.832,A 0.000,B 0.000,C 90.000,E1 5.739} C_DIS
LIN {X 0.022,Y -440.365,Z 1266.827,A 0.000,B 0.000,C 90.000,E1 4.759} C_DIS
LIN {X -0.110,Y -451.132,Z 1266.822,A 0.000,B 0.000,C 90.000,E1 3.898} C_DIS
LIN {X -0.069,Y -457.087,Z 1266.819,A 0.000,B 0.000,C 90.000,E1 3.383} C_DIS
LIN {X 0.007,Y -461.527,Z 1266.817,A 0.000,B 0.000,C 90.000,E1 2.980} C_DIS
LIN {X 0.105,Y -467.093,Z 1266.814,A 0.000,B 0.000,C 90.000,E1 2.465} C_DIS
LIN {X -0.213,Y -472.704,Z 1266.811,A 0.000,B 0.000,C 90.000,E1 1.949} C_DIS
LIN {X -0.057,Y -479.516,Z 1266.807,A 0.000,B 0.000,C 90.000,E1 1.203} C_DIS
LIN {X -0.107,Y -486.068,Z 1266.802,A 0.000,B 0.000,C 90.000,E1 0.458} C_DIS
LIN {X 0.000,Y -489.669,Z 1266.800,A 0.000,B 0.000,C 90.000,E1 360.000} C_DIS
LIN {X 0.027,Y -493.658,Z 1266.797,A 0.000,B 0.000,C 90.000,E1 359.484} C_DIS
LIN {X -0.086,Y -499.103,Z 1266.793,A 0.000,B 0.000,C 90.000,E1 358.740} C_DIS
LIN {X 0.057,Y -505.025,Z 1266.788,A 0.000,B 0.000,C 90.000,E1 357.822} C_DIS
LIN {X -0.160,Y -508.788,Z 1266.785,A 0.000,B 0.000,C 90.000,E1 357.249} C_DIS
LIN {X -0.202,Y -514.830,Z 1266.779,A 0.000,B 0.000,C 90.000,E1 356.216} C_DIS
LIN {X 0.123,Y -519.638,Z 1266.774,A 0.000,B 0.000,C 90.000,E1 355.298} C_DIS
LIN {X 0.031,Y -523.868,Z 1266.769,A 0.000,B 0.000,C 90.000,E1 354.432} C_DIS
LIN {X 0.234,Y -528.453,Z 1266.764,A 0.000,B 0.000,C 90.000,E1 353.394} C_DIS
LIN {X -0.038,Y -532.443,Z 1266.758,A 0.000,B 0.000,C 90.000,E1 352.413} C_DIS
LIN {X 0.010,Y -535.608,Z 1266.753,A 0.000,B 0.000,C 90.000,E1 351.546} C_DIS
LIN {X 0.091,Y -538.454,Z 1266.748,A 0.000,B 0.000,C 90.000,E1 350.679} C_DIS
LIN {X 0.219,Y -540.275,Z 1266.745,A 0.000,B 0.000,C 90.000,E1 350.095} C_DIS
LIN {X -0.089,Y -542.681,Z 1266.740,A 0.000,B 0.000,C 90.000,E1 349.275} C_DIS
LIN {X 0.143,Y -545.657,Z 1266.734,A 0.000,B 0.000,C 90.000,E1 348.117} C_DIS
LIN {X 0.208,Y -548.789,Z 1266.726,A 0.000,B 0.000,C 90.000,E1 346.700} C_DIS
LIN {X -0.120,Y -549.979,Z 1266.723,A 0.000,B 0.000,C 90.000,E1 346.172} C_DIS
LIN {X -0.086,Y -551.991,Z 1266.717,A 0.000,B 0.000,C 90.000,E1 345.046} C_DIS
LIN {X -0.137,Y -553.305,Z 1266.712,A 0.000,B 0.000,C 90.000,E1 344.212} C_DIS
LIN {X -0.062,Y -554.830,Z 1266.706,A 0.000,B 0.000,C 90.000,E1 343.087} C_DIS
LIN {X -0.051,Y -556.228,Z 1266.698,A 0.000,B 0.000,C 90.000,E1 341.692} C_DIS
LIN {X -0.067,Y -556.713,Z 1266.694,A 0.000,B 0.000,C 90.000,E1 340.859} C_DIS
LIN {X -0.007,Y -556.903,Z 1266.691,A 0.000,B 0.000,C 90.000,E1 340.296} C_DIS
LIN {X 0.166,Y -556.843,Z 1266.686,A 0.000,B 0.000,C 90.000,E1 339.444} C_DIS
LIN {X -0.184,Y -556.519,Z 1266.681,A 0.000,B 0.000,C 90.000,E1 338.646} C_DIS
LIN {X -0.023,Y -555.830,Z 1266.677,A 0.000,B 0.000,C 90.000,E1 337.794} C_DIS
LIN {X 0.047,Y -555.257,Z 1266.674,A 0.000,B 0.000,C 90.000,E1 337.230} C_DIS
LIN {X 0.179,Y -553.560,Z 1266.667,A 0.000,B 0.000,C 90.000,E1 336.102} C_DIS
LIN {X 0.012,Y -552.067,Z 1266.663,A 0.000,B 0.000,C 90.000,E1 335.281} C_DIS
LIN {X -0.170,Y -550.501,Z 1266.658,A 0.000,B 0.000,C 90.000,E1 334.460} C_DIS
LIN {X -0.119,Y -547.493,Z 1266.652,A 0.000,B 0.000,C 90.000,E1 333.332} C_DIS
LIN {X -0.111,Y -544.856,Z 1266.647,A 0.000,B 0.000,C 90.000,E1 332.487} C_DIS
LIN {X -0.127,Y -541.746,Z 1266.642,A 0.000,B 0.000,C 90.000,E1 331.641} C_DIS
LIN {X 0.219,Y -540.054,Z 1266.640,A 0.000,B 0.000,C 90.000,E1 331.179} C_DIS
LIN {X 0.142,Y -535.999,Z 1266.635,A 0.000,B 0.000,C 90.000,E1 330.333} C_DIS
LIN {X 0.163,Y -532.135,Z 1266.631,A 0.000,B 0.000,C 90.000,E1 329.616} C_DIS
LIN {X -0.037,Y -527.883,Z 1266.627,A 0.000,B 0.000,C 90.000,E1 328.918} C_DIS
LIN {X 0.082,Y -518.833,Z 1266.619,A 0.000,B 0.000,C 90.000,E1 327.454} C_DIS
LIN {X 0.035,Y -513.414,Z 1266.614,A 0.000,B 0.000,C 90.000,E1 326.580} C_DIS
LIN {X 0.210,Y -508.807,Z 1266.609,A 0.000,B 0.000,C 90.000,E1 325.674} C_DIS
LIN {X 0.117,Y -507.392,Z 1266.608,A 0.000,B 0.000,C 90.000,E1 325.388} C_DIS
LIN {X -0.272,Y -504.824,Z 1266.604,A 0.000,B 0.000,C 90.000,E1 324.689} C_DIS
LIN {X -0.073,Y -503.336,Z 1266.600,A 0.000,B 0.000,C 90.000,E1 324.069} C_DIS
LIN {X 0.005,Y -502.185,Z 1266.597,A 0.000,B 0.000,C 90.000,E1 323.463} C_DIS
LIN {X 0.062,Y -501.127,Z 1266.592,A 0.000,B 0.000,C 90.000,E1 322.557} C_DIS
LIN {X -0.106,Y -500.672,Z 1266.585,A 0.000,B 0.000,C 90.000,E1 321.376} C_DIS
LIN {X -0.049,Y -500.918,Z 1266.569,A 0.000,B 0.000,C 90.000,E1 318.366} C_DIS
LIN {X 0.179,Y -501.285,Z 1266.559,A 0.000,B 0.000,C 90.000,E1 316.539} C_DIS
LIN {X 0.238,Y -501.706,Z 1266.547,A 0.000,B 0.000,C 90.000,E1 314.433} C_DIS
LIN {X 0.032,Y -501.930,Z 1266.540,A 0.000,B 0.000,C 90.000,E1 313.257} C_DIS
LIN {X 0.126,Y -502.367,Z 1266.529,A 0.000,B 0.000,C 90.000,E1 311.148} C_DIS
LIN {X 0.181,Y -502.581,Z 1266.520,A 0.000,B 0.000,C 90.000,E1 309.644} C_DIS
LIN {X 0.000,Y -502.923,Z 1266.509,A 0.000,B 0.000,C 90.000,E1 307.569} C_DIS
LIN {X -0.050,Y -503.215,Z 1266.502,A 0.000,B 0.000,C 90.000,E1 306.377} C_DIS
LIN {X -0.314,Y -503.391,Z 1266.492,A 0.000,B 0.000,C 90.000,E1 304.612} C_DIS
LIN {X 0.064,Y -503.408,Z 1266.485,A 0.000,B 0.000,C 90.000,E1 303.372} C_DIS
LIN {X 0.052,Y -503.315,Z 1266.477,A 0.000,B 0.000,C 90.000,E1 301.878} C_DIS
LIN {X 0.084,Y -503.035,Z 1266.467,A 0.000,B 0.000,C 90.000,E1 300.079} C_DIS
LIN {X -0.201,Y -502.921,Z 1266.459,A 0.000,B 0.000,C 90.000,E1 298.615} C_DIS
LIN {X 0.085,Y -502.657,Z 1266.452,A 0.000,B 0.000,C 90.000,E1 297.385} C_DIS
LIN {X 0.052,Y -501.858,Z 1266.442,A 0.000,B 0.000,C 90.000,E1 295.591} C_DIS
LIN {X 0.024,Y -501.175,Z 1266.437,A 0.000,B 0.000,C 90.000,E1 294.695} C_DIS
LIN {X 0.167,Y -500.569,Z 1266.434,A 0.000,B 0.000,C 90.000,E1 294.079} C_DIS
LIN {X -0.150,Y -499.666,Z 1266.431,A 0.000,B 0.000,C 90.000,E1 293.515} C_DIS
LIN {X -0.080,Y -499.084,Z 1266.429,A 0.000,B 0.000,C 90.000,E1 293.206} C_DIS
LIN {X -0.013,Y -498.359,Z 1266.427,A 0.000,B 0.000,C 90.000,E1 292.898} C_DIS
LIN {X 0.116,Y -496.297,Z 1266.424,A 0.000,B 0.000,C 90.000,E1 292.280} C_DIS
LIN {X -0.086,Y -485.369,Z 1266.405,A 0.000,B 0.000,C 90.000,E1 288.960} C_DIS
LIN {X 0.007,Y -475.691,Z 1266.385,A 0.000,B 0.000,C 90.000,E1 285.245} C_DIS
LIN {X 0.212,Y -467.239,Z 1266.360,A 0.000,B 0.000,C 90.000,E1 280.838} C_DIS
LIN {X -0.243,Y -460.942,Z 1266.330,A 0.000,B 0.000,C 90.000,E1 275.511} C_DIS
LIN {X 0.246,Y -463.531,Z 1266.256,A 0.000,B 0.000,C 90.000,E1 262.064} C_DIS
LIN {X 0.041,Y -470.765,Z 1266.230,A 0.000,B 0.000,C 90.000,E1 257.353} C_DIS
LIN {X 0.128,Y -474.586,Z 1266.219,A 0.000,B 0.000,C 90.000,E1 255.463} C_DIS
LIN {X -0.088,Y -475.395,Z 1266.216,A 0.000,B 0.000,C 90.000,E1 254.866} C_DIS
LIN {X 0.164,Y -475.851,Z 1266.212,A 0.000,B 0.000,C 90.000,E1 254.212} C_DIS
LIN {X -0.206,Y -476.149,Z 1266.207,A 0.000,B 0.000,C 90.000,E1 253.323} C_DIS
LIN {X 0.019,Y -476.156,Z 1266.202,A 0.000,B 0.000,C 90.000,E1 252.362} C_DIS
LIN {X 0.215,Y -475.970,Z 1266.195,A 0.000,B 0.000,C 90.000,E1 251.094} C_DIS
LIN {X -0.016,Y -475.660,Z 1266.190,A 0.000,B 0.000,C 90.000,E1 250.188} C_DIS
LIN {X 0.252,Y -474.591,Z 1266.178,A 0.000,B 0.000,C 90.000,E1 247.975} C_DIS
LIN {X 0.233,Y -473.283,Z 1266.166,A 0.000,B 0.000,C 90.000,E1 245.793} C_DIS
LIN {X -0.141,Y -472.510,Z 1266.159,A 0.000,B 0.000,C 90.000,E1 244.588} C_DIS
LIN {X 0.061,Y -471.440,Z 1266.150,A 0.000,B 0.000,C 90.000,E1 242.999} C_DIS
LIN {X -0.023,Y -470.362,Z 1266.140,A 0.000,B 0.000,C 90.000,E1 241.129} C_DIS
LIN {X -0.083,Y -469.211,Z 1266.129,A 0.000,B 0.000,C 90.000,E1 239.253} C_DIS
LIN {X -0.161,Y -467.778,Z 1266.119,A 0.000,B 0.000,C 90.000,E1 237.375} C_DIS
LIN {X 0.141,Y -465.934,Z 1266.105,A 0.000,B 0.000,C 90.000,E1 234.815} C_DIS
LIN {X -0.027,Y -465.001,Z 1266.096,A 0.000,B 0.000,C 90.000,E1 233.256} C_DIS
LIN {X 0.137,Y -463.474,Z 1266.078,A 0.000,B 0.000,C 90.000,E1 230.070} C_DIS
LIN {X 0.178,Y -462.806,Z 1266.068,A 0.000,B 0.000,C 90.000,E1 228.162} C_DIS
LIN {X 0.022,Y -462.472,Z 1266.063,A 0.000,B 0.000,C 90.000,E1 227.229} C_DIS
LIN {X 0.016,Y -461.786,Z 1266.052,A 0.000,B 0.000,C 90.000,E1 225.324} C_DIS
LIN {X -0.046,Y -460.824,Z 1266.031,A 0.000,B 0.000,C 90.000,E1 221.515} C_DIS
LIN {X -0.089,Y -461.477,Z 1266.013,A 0.000,B 0.000,C 90.000,E1 218.338} C_DIS
LIN {X -0.207,Y -465.887,Z 1265.978,A 0.000,B 0.000,C 90.000,E1 212.005} C_DIS
LIN {X -0.113,Y -469.181,Z 1265.962,A 0.000,B 0.000,C 90.000,E1 209.155} C_DIS
LIN {X -0.167,Y -470.999,Z 1265.953,A 0.000,B 0.000,C 90.000,E1 207.590} C_DIS
LIN {X -0.149,Y -474.584,Z 1265.938,A 0.000,B 0.000,C 90.000,E1 204.771} C_DIS
LIN {X -0.133,Y -477.932,Z 1265.925,A 0.000,B 0.000,C 90.000,E1 202.589} C_DIS
LIN {X -0.216,Y -482.623,Z 1265.910,A 0.000,B 0.000,C 90.000,E1 199.812} C_DIS
LIN {X -0.046,Y -486.622,Z 1265.898,A 0.000,B 0.000,C 90.000,E1 197.638} C_DIS
LIN {X 0.070,Y -490.270,Z 1265.888,A 0.000,B 0.000,C 90.000,E1 195.788} C_DIS
LIN {X -0.029,Y -495.742,Z 1265.873,A 0.000,B 0.000,C 90.000,E1 193.063} C_DIS
LIN {X 0.047,Y -499.568,Z 1265.863,A 0.000,B 0.000,C 90.000,E1 191.243} C_DIS
LIN {X 0.019,Y -503.400,Z 1265.853,A 0.000,B 0.000,C 90.000,E1 189.443} C_DIS
LIN {X 0.084,Y -507.252,Z 1265.843,A 0.000,B 0.000,C 90.000,E1 187.644} C_DIS
LIN {X -0.195,Y -509.876,Z 1265.836,A 0.000,B 0.000,C 90.000,E1 186.486} C_DIS
LIN {X 0.011,Y -512.490,Z 1265.829,A 0.000,B 0.000,C 90.000,E1 185.277} C_DIS
LIN {X 0.177,Y -515.613,Z 1265.821,A 0.000,B 0.000,C 90.000,E1 183.784} C_DIS
LIN {X -0.206,Y -519.311,Z 1265.811,A 0.000,B 0.000,C 90.000,E1 182.064} C_DIS
LIN {X 0.110,Y -521.617,Z 1265.805,A 0.000,B 0.000,C 90.000,E1 180.859} C_DIS
LIN {X -0.115,Y -524.537,Z 1265.797,A 0.000,B 0.000,C 90.000,E1 179.427} C_DIS
LIN {X 0.250,Y -527.383,Z 1265.789,A 0.000,B 0.000,C 90.000,E1 177.936} C_DIS
LIN {X 0.167,Y -529.441,Z 1265.782,A 0.000,B 0.000,C 90.000,E1 176.788} C_DIS
LIN {X 0.132,Y -530.926,Z 1265.777,A 0.000,B 0.000,C 90.000,E1 175.927} C_DIS
LIN {X 0.122,Y -533.079,Z 1265.770,A 0.000,B 0.000,C 90.000,E1 174.489} C_DIS
LIN {X 0.160,Y -534.700,Z 1265.763,A 0.000,B 0.000,C 90.000,E1 173.337} C_DIS
LIN {X 0.265,Y -536.399,Z 1265.755,A 0.000,B 0.000,C 90.000,E1 171.894} C_DIS
LIN {X -0.055,Y -537.859,Z 1265.747,A 0.000,B 0.000,C 90.000,E1 170.500} C_DIS
LIN {X 0.177,Y -539.049,Z 1265.739,A 0.000,B 0.000,C 90.000,E1 169.050} C_DIS
LIN {X -0.073,Y -539.736,Z 1265.733,A 0.000,B 0.000,C 90.000,E1 167.937} C_DIS
LIN {X -0.317,Y -540.320,Z 1265.727,A 0.000,B 0.000,C 90.000,E1 166.825} C_DIS
LIN {X 0.168,Y -540.955,Z 1265.719,A 0.000,B 0.000,C 90.000,E1 165.353} C_DIS
LIN {X -0.178,Y -542.375,Z 1265.705,A 0.000,B 0.000,C 90.000,E1 162.834} C_DIS
LIN {X -0.035,Y -543.905,Z 1265.697,A 0.000,B 0.000,C 90.000,E1 161.402} C_DIS
LIN {X 0.236,Y -545.698,Z 1265.690,A 0.000,B 0.000,C 90.000,E1 160.242} C_DIS
LIN {X 0.030,Y -548.297,Z 1265.684,A 0.000,B 0.000,C 90.000,E1 159.135} C_DIS
LIN {X -0.138,Y -551.694,Z 1265.678,A 0.000,B 0.000,C 90.000,E1 158.028} C_DIS
LIN {X -0.262,Y -556.008,Z 1265.672,A 0.000,B 0.000,C 90.000,E1 156.922} C_DIS
LIN {X 0.213,Y -559.331,Z 1265.668,A 0.000,B 0.000,C 90.000,E1 156.177} C_DIS
LIN {X 0.240,Y -567.093,Z 1265.660,A 0.000,B 0.000,C 90.000,E1 154.793} C_DIS
LIN {X -0.081,Y -578.793,Z 1265.650,A 0.000,B 0.000,C 90.000,E1 153.050} C_DIS
LIN {X -0.046,Y -585.468,Z 1265.645,A 0.000,B 0.000,C 90.000,E1 152.103} C_DIS
LIN {X -0.233,Y -592.734,Z 1265.639,A 0.000,B 0.000,C 90.000,E1 151.051} C_DIS
LIN {X -0.320,Y -599.813,Z 1265.633,A 0.000,B 0.000,C 90.000,E1 149.999} C_DIS
LIN {X -0.282,Y -605.688,Z 1265.628,A 0.000,B 0.000,C 90.000,E1 149.076} C_DIS
LIN {X 0.119,Y -612.188,Z 1265.622,A 0.000,B 0.000,C 90.000,E1 147.995} C_DIS
LIN {X -0.182,Y -616.088,Z 1265.619,A 0.000,B 0.000,C 90.000,E1 147.375} C_DIS
LIN {X 0.379,Y -621.243,Z 1265.614,A 0.000,B 0.000,C 90.000,E1 146.421} C_DIS
LIN {X 0.145,Y -625.298,Z 1265.609,A 0.000,B 0.000,C 90.000,E1 145.674} C_DIS
LIN {X -0.052,Y -628.480,Z 1265.606,A 0.000,B 0.000,C 90.000,E1 145.055} C_DIS
LIN {X -0.221,Y -630.365,Z 1265.604,A 0.000,B 0.000,C 90.000,E1 144.689} C_DIS
LIN {X 0.360,Y -634.937,Z 1265.598,A 0.000,B 0.000,C 90.000,E1 143.623} C_DIS
LIN {X 0.109,Y -638.902,Z 1265.593,A 0.000,B 0.000,C 90.000,E1 142.637} C_DIS
LIN {X -0.109,Y -641.723,Z 1265.588,A 0.000,B 0.000,C 90.000,E1 141.904} C_DIS
LIN {X -0.298,Y -644.337,Z 1265.584,A 0.000,B 0.000,C 90.000,E1 141.170} C_DIS
LIN {X -0.043,Y -647.581,Z 1265.579,A 0.000,B 0.000,C 90.000,E1 140.150} C_DIS
LIN {X 0.178,Y -650.555,Z 1265.573,A 0.000,B 0.000,C 90.000,E1 139.138} C_DIS
LIN {X 0.017,Y -653.471,Z 1265.568,A 0.000,B 0.000,C 90.000,E1 138.162} C_DIS
LIN {X -0.156,Y -656.950,Z 1265.561,A 0.000,B 0.000,C 90.000,E1 136.944} C_DIS
LIN {X -0.402,Y -664.613,Z 1265.546,A 0.000,B 0.000,C 90.000,E1 134.271} C_DIS
LIN {X 0.064,Y -668.932,Z 1265.538,A 0.000,B 0.000,C 90.000,E1 132.771} C_DIS
LIN {X 0.152,Y -672.501,Z 1265.531,A 0.000,B 0.000,C 90.000,E1 131.553} C_DIS
LIN {X -0.090,Y -677.343,Z 1265.522,A 0.000,B 0.000,C 90.000,E1 129.886} C_DIS
LIN {X 0.125,Y -680.616,Z 1265.515,A 0.000,B 0.000,C 90.000,E1 128.669} C_DIS
LIN {X -0.075,Y -683.181,Z 1265.510,A 0.000,B 0.000,C 90.000,E1 127.729} C_DIS
LIN {X 0.338,Y -686.247,Z 1265.503,A 0.000,B 0.000,C 90.000,E1 126.503} C_DIS
LIN {X 0.395,Y -689.154,Z 1265.496,A 0.000,B 0.000,C 90.000,E1 125.311} C_DIS
LIN {X -0.101,Y -691.343,Z 1265.491,A 0.000,B 0.000,C 90.000,E1 124.405} C_DIS
LIN {X 0.031,Y -693.786,Z 1265.485,A 0.000,B 0.000,C 90.000,E1 123.214} C_DIS
LIN {X 0.054,Y -696.593,Z 1265.477,A 0.000,B 0.000,C 90.000,E1 121.799} C_DIS
LIN {X 0.119,Y -698.771,Z 1265.470,A 0.000,B 0.000,C 90.000,E1 120.620} C_DIS
LIN {X -0.033,Y -700.519,Z 1265.464,A 0.000,B 0.000,C 90.000,E1 119.461} C_DIS
LIN {X -0.181,Y -701.816,Z 1265.458,A 0.000,B 0.000,C 90.000,E1 118.537} C_DIS
LIN {X -0.303,Y -702.646,Z 1265.455,A 0.000,B 0.000,C 90.000,E1 117.847} C_DIS
LIN {X 0.198,Y -703.476,Z 1265.449,A 0.000,B 0.000,C 90.000,E1 116.873} C_DIS
LIN {X 0.108,Y -703.715,Z 1265.446,A 0.000,B 0.000,C 90.000,E1 116.181} C_DIS
LIN {X 0.328,Y -703.678,Z 1265.442,A 0.000,B 0.000,C 90.000,E1 115.463} C_DIS
LIN {X -0.041,Y -703.451,Z 1265.439,A 0.000,B 0.000,C 90.000,E1 115.027} C_DIS
LIN {X -0.116,Y -703.007,Z 1265.437,A 0.000,B 0.000,C 90.000,E1 114.567} C_DIS
LIN {X 0.152,Y -702.214,Z 1265.434,A 0.000,B 0.000,C 90.000,E1 114.079} C_DIS
LIN {X -0.221,Y -700.499,Z 1265.431,A 0.000,B 0.000,C 90.000,E1 113.643} C_DIS
LIN {X 0.051,Y -699.477,Z 1265.430,A 0.000,B 0.000,C 90.000,E1 113.387} C_DIS
LIN {X 0.043,Y -697.569,Z 1265.429,A 0.000,B 0.000,C 90.000,E1 113.153} C_DIS
LIN {X -0.211,Y -694.445,Z 1265.427,A 0.000,B 0.000,C 90.000,E1 112.823} C_DIS
LIN {X -0.086,Y -692.877,Z 1265.426,A 0.000,B 0.000,C 90.000,E1 112.695} C_DIS
LIN {X -0.045,Y -690.693,Z 1265.426,A 0.000,B 0.000,C 90.000,E1 112.589} C_DIS
LIN {X 0.261,Y -688.219,Z 1265.425,A 0.000,B 0.000,C 90.000,E1 112.461} C_DIS
LIN {X 0.078,Y -686.036,Z 1265.425,A 0.000,B 0.000,C 90.000,E1 112.408} C_DIS
LIN {X -0.265,Y -679.830,Z 1265.424,A 0.000,B 0.000,C 90.000,E1 112.280} C_DIS
LIN {X 0.128,Y -677.376,Z 1265.423,A 0.000,B 0.000,C 90.000,E1 112.206} C_DIS
LIN {X -0.301,Y -670.502,Z 1265.423,A 0.000,B 0.000,C 90.000,E1 112.206} C_DIS
LIN {X 0.239,Y -633.346,Z 1265.423,A 0.000,B 0.000,C 90.000,E1 112.153} C_DIS
LIN {X 0.172,Y -630.984,Z 1265.423,A 0.000,B 0.000,C 90.000,E1 112.078} C_DIS
LIN {X 0.109,Y -630.902,Z 1265.423,A 0.000,B 0.000,C 90.000,E1 112.078} C_DIS
LIN {X -0.131,Y -630.330,Z 1265.422,A 0.000,B 0.000,C 90.000,E1 112.025} C_DIS
LIN {X -0.174,Y -630.311,Z 1265.422,A 0.000,B 0.000,C 90.000,E1 112.025} C_DIS
LIN {X -0.231,Y -630.484,Z 1265.421,A 0.000,B 0.000,C 90.000,E1 111.844} C_DIS
LIN {X -0.217,Y -633.954,Z 1265.418,A 0.000,B 0.000,C 90.000,E1 111.227} C_DIS
LIN {X -0.062,Y -639.646,Z 1265.413,A 0.000,B 0.000,C 90.000,E1 110.355} C_DIS
LIN {X -0.059,Y -642.659,Z 1265.411,A 0.000,B 0.000,C 90.000,E1 109.885} C_DIS
LIN {X -0.119,Y -646.868,Z 1265.406,A 0.000,B 0.000,C 90.000,E1 109.141} C_DIS
LIN {X 0.125,Y -651.809,Z 1265.401,A 0.000,B 0.000,C 90.000,E1 108.127} C_DIS
LIN {X -0.064,Y -655.321,Z 1265.397,A 0.000,B 0.000,C 90.000,E1 107.402} C_DIS
LIN {X -0.226,Y -658.601,Z 1265.393,A 0.000,B 0.000,C 90.000,E1 106.677} C_DIS
LIN {X -0.336,Y -659.663,Z 1265.391,A 0.000,B 0.000,C 90.000,E1 106.441} C_DIS
LIN {X 0.174,Y -662.398,Z 1265.387,A 0.000,B 0.000,C 90.000,E1 105.662} C_DIS
LIN {X -0.015,Y -664.033,Z 1265.384,A 0.000,B 0.000,C 90.000,E1 105.190} C_DIS
LIN {X -0.276,Y -666.035,Z 1265.380,A 0.000,B 0.000,C 90.000,E1 104.481} C_DIS
LIN {X 0.209,Y -667.062,Z 1265.378,A 0.000,B 0.000,C 90.000,E1 103.953} C_DIS
LIN {X -0.021,Y -668.203,Z 1265.374,A 0.000,B 0.000,C 90.000,E1 103.244} C_DIS
LIN {X -0.168,Y -668.713,Z 1265.371,A 0.000,B 0.000,C 90.000,E1 102.771} C_DIS
LIN {X -0.315,Y -668.948,Z 1265.368,A 0.000,B 0.000,C 90.000,E1 102.299} C_DIS
LIN {X 0.119,Y -668.891,Z 1265.364,A 0.000,B 0.000,C 90.000,E1 101.535} C_DIS
LIN {X -0.160,Y -668.555,Z 1265.361,A 0.000,B 0.000,C 90.000,E1 101.074} C_DIS
LIN {X 0.265,Y -667.544,Z 1265.357,A 0.000,B 0.000,C 90.000,E1 100.310} C_DIS
LIN {X -0.015,Y -666.694,Z 1265.355,A 0.000,B 0.000,C 90.000,E1 99.849} C_DIS
LIN {X -0.188,Y -665.506,Z 1265.352,A 0.000,B 0.000,C 90.000,E1 99.378} C_DIS
LIN {X 0.179,Y -663.932,Z 1265.349,A 0.000,B 0.000,C 90.000,E1 98.859} C_DIS
LIN {X -0.114,Y -661.966,Z 1265.347,A 0.000,B 0.000,C 90.000,E1 98.398} C_DIS
LIN {X 0.327,Y -659.711,Z 1265.344,A 0.000,B 0.000,C 90.000,E1 97.871} C_DIS
LIN {X -0.098,Y -656.501,Z 1265.341,A 0.000,B 0.000,C 90.000,E1 97.296} C_DIS
LIN {X 0.104,Y -652.719,Z 1265.337,A 0.000,B 0.000,C 90.000,E1 96.663} C_DIS
LIN {X 0.274,Y -648.297,Z 1265.334,A 0.000,B 0.000,C 90.000,E1 96.030} C_DIS
LIN {X -0.115,Y -644.442,Z 1265.331,A 0.000,B 0.000,C 90.000,E1 95.568} C_DIS
LIN {X 0.110,Y -640.106,Z 1265.328,A 0.000,B 0.000,C 90.000,E1 95.049} C_DIS
LIN {X 0.180,Y -634.110,Z 1265.325,A 0.000,B 0.000,C 90.000,E1 94.416} C_DIS
LIN {X -0.140,Y -629.086,Z 1265.322,A 0.000,B 0.000,C 90.000,E1 93.955} C_DIS
LIN {X 0.259,Y -623.795,Z 1265.319,A 0.000,B 0.000,C 90.000,E1 93.440} C_DIS
LIN {X -0.288,Y -615.288,Z 1265.316,A 0.000,B 0.000,C 90.000,E1 92.808} C_DIS
LIN {X 0.041,Y -607.941,Z 1265.313,A 0.000,B 0.000,C 90.000,E1 92.236} C_DIS
LIN {X -0.141,Y -601.918,Z 1265.310,A 0.000,B 0.000,C 90.000,E1 91.835} C_DIS
LIN {X -0.104,Y -595.726,Z 1265.308,A 0.000,B 0.000,C 90.000,E1 91.432} C_DIS
LIN {X -0.258,Y -589.072,Z 1265.306,A 0.000,B 0.000,C 90.000,E1 91.088} C_DIS
LIN {X 0.023,Y -582.125,Z 1265.304,A 0.000,B 0.000,C 90.000,E1 90.745} C_DIS
LIN {X 0.240,Y -576.703,Z 1265.303,A 0.000,B 0.000,C 90.000,E1 90.516} C_DIS
LIN {X -0.017,Y -572.242,Z 1265.302,A 0.000,B 0.000,C 90.000,E1 90.344} C_DIS
LIN {X -0.100,Y -571.220,Z 1265.302,A 0.000,B 0.000,C 90.000,E1 90.286} C_DIS
LIN {X -0.220,Y -569.000,Z 1265.301,A 0.000,B 0.000,C 90.000,E1 90.115} C_DIS
LIN {X -0.251,Y -568.633,Z 1265.300,A 0.000,B 0.000,C 90.000,E1 90.057} C_DIS
LIN {X 0.231,Y -568.396,Z 1265.300,A 0.000,B 0.000,C 90.000,E1 89.885} C_DIS
LIN {X -0.263,Y -568.012,Z 1265.297,A 0.000,B 0.000,C 90.000,E1 89.427} C_DIS
LIN {X -0.175,Y -569.434,Z 1265.285,A 0.000,B 0.000,C 90.000,E1 87.364} C_DIS
LIN {X 0.198,Y -571.207,Z 1265.275,A 0.000,B 0.000,C 90.000,E1 85.412} C_DIS
LIN {X -0.037,Y -572.879,Z 1265.266,A 0.000,B 0.000,C 90.000,E1 83.799} C_DIS
LIN {X 0.017,Y -574.083,Z 1265.260,A 0.000,B 0.000,C 90.000,E1 82.704} C_DIS
LIN {X -0.086,Y -575.875,Z 1265.250,A 0.000,B 0.000,C 90.000,E1 81.084} C_DIS
LIN {X -0.273,Y -577.244,Z 1265.243,A 0.000,B 0.000,C 90.000,E1 79.746} C_DIS
LIN {X 0.023,Y -578.160,Z 1265.237,A 0.000,B 0.000,C 90.000,E1 78.634} C_DIS
LIN {X 0.214,Y -579.435,Z 1265.228,A 0.000,B 0.000,C 90.000,E1 76.992} C_DIS
LIN {X -0.144,Y -580.600,Z 1265.219,A 0.000,B 0.000,C 90.000,E1 75.408} C_DIS
LIN {X 0.110,Y -581.146,Z 1265.214,A 0.000,B 0.000,C 90.000,E1 74.574} C_DIS
LIN {X -0.307,Y -581.921,Z 1265.207,A 0.000,B 0.000,C 90.000,E1 73.268} C_DIS
LIN {X -0.150,Y -582.906,Z 1265.198,A 0.000,B 0.000,C 90.000,E1 71.638} C_DIS
LIN {X -0.178,Y -583.716,Z 1265.190,A 0.000,B 0.000,C 90.000,E1 70.296} C_DIS
LIN {X -0.257,Y -584.925,Z 1265.179,A 0.000,B 0.000,C 90.000,E1 68.156} C_DIS
LIN {X -0.348,Y -586.991,Z 1265.164,A 0.000,B 0.000,C 90.000,E1 65.485} C_DIS
LIN {X 0.134,Y -588.073,Z 1265.156,A 0.000,B 0.000,C 90.000,E1 64.101} C_DIS
LIN {X 0.038,Y -589.910,Z 1265.144,A 0.000,B 0.000,C 90.000,E1 61.975} C_DIS
LIN {X -0.136,Y -591.796,Z 1265.134,A 0.000,B 0.000,C 90.000,E1 60.127} C_DIS
LIN {X 0.045,Y -593.740,Z 1265.124,A 0.000,B 0.000,C 90.000,E1 58.250} C_DIS
LIN {X 0.153,Y -595.090,Z 1265.116,A 0.000,B 0.000,C 90.000,E1 56.914} C_DIS
LIN {X 0.107,Y -596.444,Z 1265.109,A 0.000,B 0.000,C 90.000,E1 55.595} C_DIS
LIN {X 0.082,Y -597.644,Z 1265.102,A 0.000,B 0.000,C 90.000,E1 54.276} C_DIS
LIN {X 0.186,Y -598.978,Z 1265.093,A 0.000,B 0.000,C 90.000,E1 52.683} C_DIS
LIN {X 0.322,Y -600.219,Z 1265.084,A 0.000,B 0.000,C 90.000,E1 51.090} C_DIS
LIN {X -0.259,Y -600.801,Z 1265.080,A 0.000,B 0.000,C 90.000,E1 50.356} C_DIS
LIN {X 0.008,Y -601.168,Z 1265.075,A 0.000,B 0.000,C 90.000,E1 49.542} C_DIS
LIN {X 0.089,Y -601.761,Z 1265.067,A 0.000,B 0.000,C 90.000,E1 47.957} C_DIS
LIN {X 0.110,Y -602.176,Z 1265.061,A 0.000,B 0.000,C 90.000,E1 46.905} C_DIS
LIN {X -0.269,Y -602.437,Z 1265.055,A 0.000,B 0.000,C 90.000,E1 45.891} C_DIS
LIN {X -0.226,Y -602.541,Z 1265.049,A 0.000,B 0.000,C 90.000,E1 44.838} C_DIS
LIN {X -0.184,Y -602.413,Z 1265.043,A 0.000,B 0.000,C 90.000,E1 43.785} C_DIS
LIN {X 0.290,Y -602.110,Z 1265.037,A 0.000,B 0.000,C 90.000,E1 42.690} C_DIS
LIN {X 0.149,Y -601.621,Z 1265.030,A 0.000,B 0.000,C 90.000,E1 41.391} C_DIS
LIN {X -0.001,Y -601.047,Z 1265.023,A 0.000,B 0.000,C 90.000,E1 40.092} C_DIS
LIN {X 0.293,Y -600.232,Z 1265.016,A 0.000,B 0.000,C 90.000,E1 38.749} C_DIS
LIN {X -0.047,Y -599.451,Z 1265.010,A 0.000,B 0.000,C 90.000,E1 37.729} C_DIS
LIN {X -0.161,Y -598.637,Z 1265.005,A 0.000,B 0.000,C 90.000,E1 36.950} C_DIS
LIN {X -0.041,Y -597.345,Z 1264.999,A 0.000,B 0.000,C 90.000,E1 35.884} C_DIS
LIN {X 0.055,Y -595.789,Z 1264.994,A 0.000,B 0.000,C 90.000,E1 34.818} C_DIS
LIN {X -0.099,Y -594.329,Z 1264.989,A 0.000,B 0.000,C 90.000,E1 34.040} C_DIS
LIN {X 0.109,Y -592.159,Z 1264.983,A 0.000,B 0.000,C 90.000,E1 32.959} C_DIS
LIN {X 0.204,Y -590.951,Z 1264.980,A 0.000,B 0.000,C 90.000,E1 32.418} C_DIS
LIN {X -0.134,Y -587.995,Z 1264.974,A 0.000,B 0.000,C 90.000,E1 31.386} C_DIS
LIN {X -0.193,Y -585.363,Z 1264.970,A 0.000,B 0.000,C 90.000,E1 30.590} C_DIS
LIN {X -0.149,Y -583.446,Z 1264.967,A 0.000,B 0.000,C 90.000,E1 30.050} C_DIS
LIN {X 0.251,Y -580.088,Z 1264.962,A 0.000,B 0.000,C 90.000,E1 29.205} C_DIS
LIN {X -0.025,Y -577.628,Z 1264.959,A 0.000,B 0.000,C 90.000,E1 28.693} C_DIS
LIN {X -0.045,Y -575.016,Z 1264.956,A 0.000,B 0.000,C 90.000,E1 28.153} C_DIS
LIN {X 0.153,Y -572.150,Z 1264.953,A 0.000,B 0.000,C 90.000,E1 27.590} C_DIS
LIN {X 0.087,Y -569.078,Z 1264.950,A 0.000,B 0.000,C 90.000,E1 27.052} C_DIS
LIN {X 0.155,Y -564.913,Z 1264.947,A 0.000,B 0.000,C 90.000,E1 26.360} C_DIS
LIN {X 0.093,Y -559.544,Z 1264.942,A 0.000,B 0.000,C 90.000,E1 25.540} C_DIS
LIN {X 0.144,Y -554.628,Z 1264.938,A 0.000,B 0.000,C 90.000,E1 24.847} C_DIS
LIN {X -0.296,Y -550.366,Z 1264.935,A 0.000,B 0.000,C 90.000,E1 24.335} C_DIS
LIN {X -0.240,Y -543.743,Z 1264.931,A 0.000,B 0.000,C 90.000,E1 23.515} C_DIS
LIN {X 0.122,Y -537.642,Z 1264.927,A 0.000,B 0.000,C 90.000,E1 22.770} C_DIS
LIN {X -0.086,Y -527.726,Z 1264.921,A 0.000,B 0.000,C 90.000,E1 21.716} C_DIS
LIN {X 0.081,Y -518.486,Z 1264.915,A 0.000,B 0.000,C 90.000,E1 20.737} C_DIS
LIN {X 0.190,Y -507.711,Z 1264.909,A 0.000,B 0.000,C 90.000,E1 19.631} C_DIS
LIN {X 0.152,Y -495.018,Z 1264.902,A 0.000,B 0.000,C 90.000,E1 18.417} C_DIS
LIN {X -0.054,Y -485.066,Z 1264.897,A 0.000,B 0.000,C 90.000,E1 17.511} C_DIS
LIN {X -0.154,Y -477.651,Z 1264.894,A 0.000,B 0.000,C 90.000,E1 16.858} C_DIS
LIN {X 0.088,Y -465.859,Z 1264.888,A 0.000,B 0.000,C 90.000,E1 15.788} C_DIS
LIN {X 0.225,Y -445.229,Z 1264.877,A 0.000,B 0.000,C 90.000,E1 13.883} C_DIS
LIN {X 0.014,Y -423.655,Z 1264.865,A 0.000,B 0.000,C 90.000,E1 11.771} C_DIS
LIN {X 0.084,Y -406.502,Z 1264.855,A 0.000,B 0.000,C 90.000,E1 9.905} C_DIS
LIN {X -0.049,Y -399.887,Z 1264.851,A 0.000,B 0.000,C 90.000,E1 9.151} C_DIS
LIN {X 0.084,Y -398.591,Z 1264.850,A 0.000,B 0.000,C 90.000,E1 8.973} C_DIS
LIN {X 0.066,Y -394.906,Z 1264.847,A 0.000,B 0.000,C 90.000,E1 8.398} C_DIS
LIN {X 0.029,Y -394.880,Z 1264.847,A 0.000,B 0.000,C 90.000,E1 8.398} C_DIS
LIN {X 0.116,Y -394.779,Z 1264.846,A 0.000,B 0.000,C 90.000,E1 8.341} C_DIS
LIN {X 0.078,Y -394.788,Z 1264.846,A 0.000,B 0.000,C 90.000,E1 8.341} C_DIS
LIN {X 0.064,Y -395.578,Z 1264.845,A 0.000,B 0.000,C 90.000,E1 8.106} C_DIS
LIN {X -0.155,Y -396.045,Z 1264.845,A 0.000,B 0.000,C 90.000,E1 8.049} C_DIS
LIN {X 0.012,Y -399.367,Z 1264.843,A 0.000,B 0.000,C 90.000,E1 7.701} C_DIS
LIN {X -0.203,Y -401.141,Z 1264.842,A 0.000,B 0.000,C 90.000,E1 7.587} C_DIS
LIN {X -0.115,Y -415.351,Z 1264.837,A 0.000,B 0.000,C 90.000,E1 6.663} C_DIS
LIN {X 0.007,Y -423.322,Z 1264.834,A 0.000,B 0.000,C 90.000,E1 6.087} C_DIS
LIN {X -0.153,Y -431.114,Z 1264.831,A 0.000,B 0.000,C 90.000,E1 5.511} C_DIS
LIN {X -0.130,Y -442.125,Z 1264.826,A 0.000,B 0.000,C 90.000,E1 4.645} C_DIS
LIN {X 0.059,Y -454.388,Z 1264.820,A 0.000,B 0.000,C 90.000,E1 3.612} C_DIS
LIN {X 0.077,Y -464.797,Z 1264.815,A 0.000,B 0.000,C 90.000,E1 2.694} C_DIS
LIN {X 0.114,Y -468.991,Z 1264.813,A 0.000,B 0.000,C 90.000,E1 2.293} C_DIS
LIN {X -0.027,Y -473.245,Z 1264.811,A 0.000,B 0.000,C 90.000,E1 1.892} C_DIS
LIN {X 0.195,Y -479.992,Z 1264.807,A 0.000,B 0.000,C 90.000,E1 1.146} C_DIS
LIN {X 0.123,Y -486.630,Z 1264.802,A 0.000,B 0.000,C 90.000,E1 0.401} C_DIS
LIN {X 0.000,Y -489.977,Z 1264.800,A 0.000,B 0.000,C 90.000,E1 360.000} C_DIS
LIN {X 0.028,Y -493.996,Z 1264.797,A 0.000,B 0.000,C 90.000,E1 359.484} C_DIS
LIN {X -0.081,Y -499.466,Z 1264.793,A 0.000,B 0.000,C 90.000,E1 358.740} C_DIS
LIN {X 0.066,Y -505.400,Z 1264.788,A 0.000,B 0.000,C 90.000,E1 357.822} C_DIS
LIN {X -0.149,Y -509.194,Z 1264.785,A 0.000,B 0.000,C 90.000,E1 357.249} C_DIS
LIN {X -0.185,Y -515.258,Z 1264.779,A 0.000,B 0.000,C 90.000,E1 356.216} C_DIS
LIN {X -0.079,Y -519.286,Z 1264.775,A 0.000,B 0.000,C 90.000,E1 355.469} C_DIS
LIN {X 0.065,Y -522.961,Z 1264.771,A 0.000,B 0.000,C 90.000,E1 354.723} C_DIS
LIN {X 0.251,Y -527.617,Z 1264.765,A 0.000,B 0.000,C 90.000,E1 353.685} C_DIS
LIN {X -0.017,Y -529.535,Z 1264.763,A 0.000,B 0.000,C 90.000,E1 353.280} C_DIS
LIN {X 0.001,Y -532.916,Z 1264.758,A 0.000,B 0.000,C 90.000,E1 352.413} C_DIS
LIN {X 0.055,Y -536.080,Z 1264.753,A 0.000,B 0.000,C 90.000,E1 351.546} C_DIS
LIN {X 0.204,Y -539.810,Z 1264.747,A 0.000,B 0.000,C 90.000,E1 350.387} C_DIS
LIN {X -0.187,Y -541.548,Z 1264.744,A 0.000,B 0.000,C 90.000,E1 349.859} C_DIS
LIN {X -0.051,Y -543.908,Z 1264.739,A 0.000,B 0.000,C 90.000,E1 348.993} C_DIS
LIN {X 0.209,Y -546.110,Z 1264.734,A 0.000,B 0.000,C 90.000,E1 348.117} C_DIS
LIN {X 0.179,Y -548.647,Z 1264.728,A 0.000,B 0.000,C 90.000,E1 346.992} C_DIS
LIN {X -0.042,Y -550.463,Z 1264.723,A 0.000,B 0.000,C 90.000,E1 346.172} C_DIS
LIN {X -0.001,Y -552.488,Z 1264.717,A 0.000,B 0.000,C 90.000,E1 345.046} C_DIS
LIN {X 0.067,Y -554.209,Z 1264.711,A 0.000,B 0.000,C 90.000,E1 343.921} C_DIS
LIN {X 0.316,Y -555.689,Z 1264.705,A 0.000,B 0.000,C 90.000,E1 342.779} C_DIS
LIN {X 0.058,Y -556.798,Z 1264.698,A 0.000,B 0.000,C 90.000,E1 341.692} C_DIS
LIN {X 0.047,Y -557.329,Z 1264.694,A 0.000,B 0.000,C 90.000,E1 340.859} C_DIS
LIN {X 0.220,Y -557.580,Z 1264.689,A 0.000,B 0.000,C 90.000,E1 340.007} C_DIS
LIN {X -0.128,Y -557.466,Z 1264.684,A 0.000,B 0.000,C 90.000,E1 339.209} C_DIS
LIN {X 0.043,Y -557.090,Z 1264.680,A 0.000,B 0.000,C 90.000,E1 338.358} C_DIS
LIN {X 0.194,Y -556.060,Z 1264.674,A 0.000,B 0.000,C 90.000,E1 337.230} C_DIS
LIN {X 0.268,Y -555.301,Z 1264.671,A 0.000,B 0.000,C 90.000,E1 336.666} C_DIS
LIN {X -0.109,Y -554.004,Z 1264.666,A 0.000,B 0.000,C 90.000,E1 335.869} C_DIS
LIN {X 0.005,Y -551.374,Z 1264.658,A 0.000,B 0.000,C 90.000,E1 334.460} C_DIS
LIN {X -0.188,Y -549.191,Z 1264.653,A 0.000,B 0.000,C 90.000,E1 333.640} C_DIS
LIN {X -0.158,Y -546.833,Z 1264.649,A 0.000,B 0.000,C 90.000,E1 332.794} C_DIS
LIN {X 0.331,Y -543.907,Z 1264.644,A 0.000,B 0.000,C 90.000,E1 331.897} C_DIS
LIN {X -0.303,Y -541.063,Z 1264.640,A 0.000,B 0.000,C 90.000,E1 331.257} C_DIS
LIN {X -0.102,Y -537.071,Z 1264.635,A 0.000,B 0.000,C 90.000,E1 330.383} C_DIS
LIN {X -0.210,Y -532.449,Z 1264.631,A 0.000,B 0.000,C 90.000,E1 329.537} C_DIS
LIN {X -0.072,Y -529.000,Z 1264.627,A 0.000,B 0.000,C 90.000,E1 328.948} C_DIS
LIN {X -0.052,Y -521.694,Z 1264.621,A 0.000,B 0.000,C 90.000,E1 327.788} C_DIS
LIN {X -0.248,Y -513.533,Z 1264.614,A 0.000,B 0.000,C 90.000,E1 326.501} C_DIS
LIN {X -0.130,Y -510.501,Z 1264.611,A 0.000,B 0.000,C 90.000,E1 325.928} C_DIS
LIN {X 0.068,Y -507.777,Z 1264.608,A 0.000,B 0.000,C 90.000,E1 325.341} C_DIS
LIN {X 0.077,Y -504.962,Z 1264.603,A 0.000,B 0.000,C 90.000,E1 324.529} C_DIS
LIN {X 0.279,Y -503.517,Z 1264.600,A 0.000,B 0.000,C 90.000,E1 323.909} C_DIS
LIN {X 0.060,Y -502.450,Z 1264.596,A 0.000,B 0.000,C 90.000,E1 323.336} C_DIS
LIN {X -0.166,Y -501.675,Z 1264.593,A 0.000,B 0.000,C 90.000,E1 322.763} C_DIS
LIN {X 0.068,Y -501.086,Z 1264.586,A 0.000,B 0.000,C 90.000,E1 321.537} C_DIS
LIN {X 0.007,Y -501.374,Z 1264.568,A 0.000,B 0.000,C 90.000,E1 318.243} C_DIS
LIN {X 0.005,Y -501.691,Z 1264.560,A 0.000,B 0.000,C 90.000,E1 316.743} C_DIS
LIN {X -0.271,Y -502.111,Z 1264.548,A 0.000,B 0.000,C 90.000,E1 314.676} C_DIS
LIN {X -0.127,Y -502.367,Z 1264.541,A 0.000,B 0.000,C 90.000,E1 313.461} C_DIS
LIN {X -0.031,Y -502.784,Z 1264.530,A 0.000,B 0.000,C 90.000,E1 311.353} C_DIS
LIN {X 0.026,Y -503.040,Z 1264.521,A 0.000,B 0.000,C 90.000,E1 309.850} C_DIS
LIN {X 0.138,Y -503.450,Z 1264.508,A 0.000,B 0.000,C 90.000,E1 307.443} C_DIS
LIN {X 0.100,Y -503.712,Z 1264.501,A 0.000,B 0.000,C 90.000,E1 306.251} C_DIS
LIN {X -0.036,Y -503.887,Z 1264.493,A 0.000,B 0.000,C 90.000,E1 304.771} C_DIS
LIN {X -0.065,Y -503.938,Z 1264.487,A 0.000,B 0.000,C 90.000,E1 303.579} C_DIS
LIN {X -0.066,Y -503.900,Z 1264.478,A 0.000,B 0.000,C 90.000,E1 302.084} C_DIS
LIN {X 0.234,Y -503.640,Z 1264.468,A 0.000,B 0.000,C 90.000,E1 300.256} C_DIS
LIN {X -0.290,Y -503.540,Z 1264.460,A 0.000,B 0.000,C 90.000,E1 298.821} C_DIS
LIN {X 0.010,Y -503.342,Z 1264.453,A 0.000,B 0.000,C 90.000,E1 297.590} C_DIS
LIN {X 0.295,Y -503.005,Z 1264.442,A 0.000,B 0.000,C 90.000,E1 295.463} C_DIS
LIN {X -0.310,Y -502.603,Z 1264.435,A 0.000,B 0.000,C 90.000,E1 294.335} C_DIS
LIN {X 0.126,Y -502.018,Z 1264.430,A 0.000,B 0.000,C 90.000,E1 293.387} C_DIS
LIN {X -0.107,Y -501.083,Z 1264.425,A 0.000,B 0.000,C 90.000,E1 292.514} C_DIS
LIN {X 0.112,Y -499.797,Z 1264.420,A 0.000,B 0.000,C 90.000,E1 291.589} C_DIS
LIN {X 0.249,Y -498.602,Z 1264.417,A 0.000,B 0.000,C 90.000,E1 290.972} C_DIS
LIN {X 0.139,Y -497.798,Z 1264.415,A 0.000,B 0.000,C 90.000,E1 290.684} C_DIS
LIN {X 0.165,Y -486.967,Z 1264.395,A 0.000,B 0.000,C 90.000,E1 287.040} C_DIS
LIN {X -0.063,Y -477.793,Z 1264.373,A 0.000,B 0.000,C 90.000,E1 283.063} C_DIS
LIN {X -0.163,Y -470.403,Z 1264.347,A 0.000,B 0.000,C 90.000,E1 278.398} C_DIS
LIN {X -0.121,Y -465.506,Z 1264.306,A 0.000,B 0.000,C 90.000,E1 271.146} C_DIS
LIN {X 0.143,Y -469.549,Z 1264.259,A 0.000,B 0.000,C 90.000,E1 262.591} C_DIS
LIN {X -0.205,Y -476.427,Z 1264.233,A 0.000,B 0.000,C 90.000,E1 257.937} C_DIS
LIN {X 0.101,Y -476.900,Z 1264.231,A 0.000,B 0.000,C 90.000,E1 257.589} C_DIS
LIN {X -0.109,Y -477.447,Z 1264.228,A 0.000,B 0.000,C 90.000,E1 256.992} C_DIS
LIN {X -0.149,Y -477.898,Z 1264.221,A 0.000,B 0.000,C 90.000,E1 255.755} C_DIS
LIN {X -0.189,Y -478.038,Z 1264.214,A 0.000,B 0.000,C 90.000,E1 254.519} C_DIS
LIN {X -0.108,Y -477.780,Z 1264.207,A 0.000,B 0.000,C 90.000,E1 253.268} C_DIS
LIN {X 0.110,Y -477.247,Z 1264.200,A 0.000,B 0.000,C 90.000,E1 252.000} C_DIS
LIN {X -0.146,Y -476.497,Z 1264.192,A 0.000,B 0.000,C 90.000,E1 250.477} C_DIS
LIN {X 0.030,Y -475.688,Z 1264.183,A 0.000,B 0.000,C 90.000,E1 248.901} C_DIS
LIN {X -0.064,Y -475.060,Z 1264.176,A 0.000,B 0.000,C 90.000,E1 247.667} C_DIS
LIN {X -0.041,Y -473.913,Z 1264.166,A 0.000,B 0.000,C 90.000,E1 245.793} C_DIS
LIN {X 0.022,Y -473.142,Z 1264.159,A 0.000,B 0.000,C 90.000,E1 244.537} C_DIS
LIN {X -0.190,Y -472.082,Z 1264.150,A 0.000,B 0.000,C 90.000,E1 242.999} C_DIS
LIN {X -0.033,Y -470.954,Z 1264.140,A 0.000,B 0.000,C 90.000,E1 241.101} C_DIS
LIN {X 0.098,Y -469.760,Z 1264.129,A 0.000,B 0.000,C 90.000,E1 239.203} C_DIS
LIN {X -0.134,Y -468.549,Z 1264.120,A 0.000,B 0.000,C 90.000,E1 237.661} C_DIS
LIN {X -0.228,Y -466.883,Z 1264.108,A 0.000,B 0.000,C 90.000,E1 235.468} C_DIS
LIN {X 0.163,Y -465.497,Z 1264.096,A 0.000,B 0.000,C 90.000,E1 233.210} C_DIS
LIN {X -0.027,Y -463.956,Z 1264.078,A 0.000,B 0.000,C 90.000,E1 230.070} C_DIS
LIN {X 0.026,Y -463.241,Z 1264.068,A 0.000,B 0.000,C 90.000,E1 228.162} C_DIS
LIN {X -0.179,Y -463.054,Z 1264.064,A 0.000,B 0.000,C 90.000,E1 227.553} C_DIS
LIN {X -0.122,Y -462.138,Z 1264.052,A 0.000,B 0.000,C 90.000,E1 225.324} C_DIS
LIN {X -0.169,Y -461.073,Z 1264.031,A 0.000,B 0.000,C 90.000,E1 221.515} C_DIS
LIN {X -0.172,Y -461.836,Z 1264.011,A 0.000,B 0.000,C 90.000,E1 218.016} C_DIS
LIN {X -0.054,Y -465.756,Z 1263.979,A 0.000,B 0.000,C 90.000,E1 212.291} C_DIS
LIN {X -0.130,Y -468.964,Z 1263.964,A 0.000,B 0.000,C 90.000,E1 209.461} C_DIS
LIN {X -0.197,Y -470.848,Z 1263.955,A 0.000,B 0.000,C 90.000,E1 207.897} C_DIS
LIN {X -0.229,Y -474.782,Z 1263.938,A 0.000,B 0.000,C 90.000,E1 204.771} C_DIS
LIN {X -0.209,Y -478.120,Z 1263.925,A 0.000,B 0.000,C 90.000,E1 202.589} C_DIS
LIN {X 0.168,Y -482.802,Z 1263.910,A 0.000,B 0.000,C 90.000,E1 199.758} C_DIS
LIN {X -0.112,Y -486.850,Z 1263.898,A 0.000,B 0.000,C 90.000,E1 197.638} C_DIS
LIN {X 0.010,Y -490.538,Z 1263.888,A 0.000,B 0.000,C 90.000,E1 195.788} C_DIS
LIN {X 0.013,Y -495.428,Z 1263.874,A 0.000,B 0.000,C 90.000,E1 193.355} C_DIS
LIN {X 0.081,Y -499.288,Z 1263.864,A 0.000,B 0.000,C 90.000,E1 191.535} C_DIS
LIN {X 0.133,Y -503.190,Z 1263.854,A 0.000,B 0.000,C 90.000,E1 189.726} C_DIS
LIN {X 0.112,Y -507.083,Z 1263.844,A 0.000,B 0.000,C 90.000,E1 187.936} C_DIS
LIN {X -0.164,Y -509.794,Z 1263.838,A 0.000,B 0.000,C 90.000,E1 186.777} C_DIS
LIN {X 0.001,Y -513.072,Z 1263.829,A 0.000,B 0.000,C 90.000,E1 185.277} C_DIS
LIN {X 0.178,Y -516.257,Z 1263.821,A 0.000,B 0.000,C 90.000,E1 183.784} C_DIS
LIN {X -0.191,Y -520.051,Z 1263.811,A 0.000,B 0.000,C 90.000,E1 182.064} C_DIS
LIN {X 0.137,Y -522.420,Z 1263.805,A 0.000,B 0.000,C 90.000,E1 180.859} C_DIS
LIN {X -0.073,Y -525.405,Z 1263.797,A 0.000,B 0.000,C 90.000,E1 179.427} C_DIS
LIN {X -0.220,Y -528.316,Z 1263.789,A 0.000,B 0.000,C 90.000,E1 177.993} C_DIS
LIN {X 0.239,Y -530.467,Z 1263.782,A 0.000,B 0.000,C 90.000,E1 176.788} C_DIS
LIN {X 0.199,Y -532.429,Z 1263.776,A 0.000,B 0.000,C 90.000,E1 175.641} C_DIS
LIN {X 0.210,Y -534.658,Z 1263.768,A 0.000,B 0.000,C 90.000,E1 174.204} C_DIS
LIN {X -0.267,Y -536.284,Z 1263.762,A 0.000,B 0.000,C 90.000,E1 173.109} C_DIS
LIN {X -0.123,Y -537.769,Z 1263.755,A 0.000,B 0.000,C 90.000,E1 171.951} C_DIS
LIN {X 0.114,Y -539.344,Z 1263.747,A 0.000,B 0.000,C 90.000,E1 170.500} C_DIS
LIN {X -0.228,Y -540.434,Z 1263.741,A 0.000,B 0.000,C 90.000,E1 169.398} C_DIS
LIN {X 0.071,Y -541.299,Z 1263.735,A 0.000,B 0.000,C 90.000,E1 168.229} C_DIS
LIN {X -0.071,Y -542.187,Z 1263.727,A 0.000,B 0.000,C 90.000,E1 166.825} C_DIS
LIN {X -0.227,Y -543.441,Z 1263.714,A 0.000,B 0.000,C 90.000,E1 164.574} C_DIS
LIN {X -0.198,Y -545.322,Z 1263.702,A 0.000,B 0.000,C 90.000,E1 162.308} C_DIS
LIN {X -0.159,Y -546.503,Z 1263.697,A 0.000,B 0.000,C 90.000,E1 161.456} C_DIS
LIN {X -0.030,Y -548.532,Z 1263.691,A 0.000,B 0.000,C 90.000,E1 160.315} C_DIS
LIN {X -0.204,Y -551.244,Z 1263.684,A 0.000,B 0.000,C 90.000,E1 159.209} C_DIS
LIN {X 0.103,Y -553.832,Z 1263.680,A 0.000,B 0.000,C 90.000,E1 158.337} C_DIS
LIN {X 0.234,Y -556.901,Z 1263.675,A 0.000,B 0.000,C 90.000,E1 157.486} C_DIS
LIN {X -0.108,Y -561.952,Z 1263.669,A 0.000,B 0.000,C 90.000,E1 156.410} C_DIS
LIN {X 0.061,Y -568.694,Z 1263.662,A 0.000,B 0.000,C 90.000,E1 155.153} C_DIS
LIN {X 0.098,Y -586.134,Z 1263.647,A 0.000,B 0.000,C 90.000,E1 152.436} C_DIS
LIN {X -0.083,Y -593.152,Z 1263.641,A 0.000,B 0.000,C 90.000,E1 151.385} C_DIS
LIN {X -0.124,Y -599.131,Z 1263.636,A 0.000,B 0.000,C 90.000,E1 150.461} C_DIS
LIN {X -0.091,Y -604.899,Z 1263.631,A 0.000,B 0.000,C 90.000,E1 149.537} C_DIS
LIN {X 0.301,Y -611.227,Z 1263.625,A 0.000,B 0.000,C 90.000,E1 148.456} C_DIS
LIN {X -0.025,Y -615.849,Z 1263.621,A 0.000,B 0.000,C 90.000,E1 147.709} C_DIS
LIN {X 0.211,Y -620.158,Z 1263.616,A 0.000,B 0.000,C 90.000,E1 146.914} C_DIS
LIN {X 0.303,Y -624.897,Z 1263.611,A 0.000,B 0.000,C 90.000,E1 146.008} C_DIS
LIN {X -0.053,Y -629.890,Z 1263.606,A 0.000,B 0.000,C 90.000,E1 145.022} C_DIS
LIN {X 0.301,Y -632.218,Z 1263.603,A 0.000,B 0.000,C 90.000,E1 144.482} C_DIS
LIN {X 0.014,Y -635.531,Z 1263.599,A 0.000,B 0.000,C 90.000,E1 143.749} C_DIS
LIN {X -0.107,Y -638.513,Z 1263.594,A 0.000,B 0.000,C 90.000,E1 143.004} C_DIS
LIN {X 0.069,Y -642.175,Z 1263.589,A 0.000,B 0.000,C 90.000,E1 141.984} C_DIS
LIN {X -0.116,Y -644.748,Z 1263.585,A 0.000,B 0.000,C 90.000,E1 141.251} C_DIS
LIN {X 0.143,Y -647.883,Z 1263.579,A 0.000,B 0.000,C 90.000,E1 140.231} C_DIS
LIN {X -0.058,Y -650.846,Z 1263.574,A 0.000,B 0.000,C 90.000,E1 139.256} C_DIS
LIN {X 0.163,Y -654.382,Z 1263.567,A 0.000,B 0.000,C 90.000,E1 138.000} C_DIS
LIN {X 0.041,Y -657.113,Z 1263.561,A 0.000,B 0.000,C 90.000,E1 137.025} C_DIS
LIN {X -0.177,Y -663.212,Z 1263.549,A 0.000,B 0.000,C 90.000,E1 134.838} C_DIS
LIN {X -0.220,Y -667.475,Z 1263.541,A 0.000,B 0.000,C 90.000,E1 133.380} C_DIS
LIN {X -0.164,Y -671.045,Z 1263.534,A 0.000,B 0.000,C 90.000,E1 132.162} C_DIS
LIN {X 0.388,Y -673.848,Z 1263.529,A 0.000,B 0.000,C 90.000,E1 131.148} C_DIS
LIN {X 0.141,Y -677.924,Z 1263.521,A 0.000,B 0.000,C 90.000,E1 129.725} C_DIS
LIN {X 0.337,Y -680.516,Z 1263.516,A 0.000,B 0.000,C 90.000,E1 128.749} C_DIS
LIN {X -0.250,Y -683.689,Z 1263.509,A 0.000,B 0.000,C 90.000,E1 127.604} C_DIS
LIN {X 0.176,Y -686.735,Z 1263.502,A 0.000,B 0.000,C 90.000,E1 126.377} C_DIS
LIN {X -0.318,Y -689.633,Z 1263.496,A 0.000,B 0.000,C 90.000,E1 125.231} C_DIS
LIN {X 0.119,Y -691.264,Z 1263.492,A 0.000,B 0.000,C 90.000,E1 124.485} C_DIS
LIN {X 0.254,Y -693.723,Z 1263.485,A 0.000,B 0.000,C 90.000,E1 123.293} C_DIS
LIN {X 0.281,Y -696.563,Z 1263.477,A 0.000,B 0.000,C 90.000,E1 121.878} C_DIS
LIN {X 0.106,Y -698.748,Z 1263.471,A 0.000,B 0.000,C 90.000,E1 120.718} C_DIS
LIN {X -0.060,Y -700.183,Z 1263.466,A 0.000,B 0.000,C 90.000,E1 119.795} C_DIS
LIN {X 0.063,Y -701.860,Z 1263.459,A 0.000,B 0.000,C 90.000,E1 118.615} C_DIS
LIN {X 0.274,Y -702.730,Z 1263.455,A 0.000,B 0.000,C 90.000,E1 117.897} C_DIS
LIN {X -0.175,Y -703.624,Z 1263.450,A 0.000,B 0.000,C 90.000,E1 117.001} C_DIS
LIN {X 0.046,Y -703.910,Z 1263.446,A 0.000,B 0.000,C 90.000,E1 116.283} C_DIS
LIN {X -0.326,Y -703.982,Z 1263.443,A 0.000,B 0.000,C 90.000,E1 115.848} C_DIS
LIN {X -0.410,Y -703.747,Z 1263.440,A 0.000,B 0.000,C 90.000,E1 115.155} C_DIS
LIN {X 0.158,Y -703.406,Z 1263.437,A 0.000,B 0.000,C 90.000,E1 114.643} C_DIS
LIN {X -0.211,Y -702.597,Z 1263.434,A 0.000,B 0.000,C 90.000,E1 114.207} C_DIS
LIN {X 0.069,Y -702.033,Z 1263.433,A 0.000,B 0.000,C 90.000,E1 113.951} C_DIS
LIN {X -0.305,Y -700.209,Z 1263.431,A 0.000,B 0.000,C 90.000,E1 113.515} C_DIS
LIN {X -0.170,Y -699.614,Z 1263.430,A 0.000,B 0.000,C 90.000,E1 113.387} C_DIS
LIN {X 0.096,Y -697.649,Z 1263.429,A 0.000,B 0.000,C 90.000,E1 113.131} C_DIS
LIN {X 0.210,Y -694.495,Z 1263.427,A 0.000,B 0.000,C 90.000,E1 112.770} C_DIS
LIN {X 0.334,Y -692.852,Z 1263.426,A 0.000,B 0.000,C 90.000,E1 112.642} C_DIS
LIN {X 0.223,Y -688.437,Z 1263.425,A 0.000,B 0.000,C 90.000,E1 112.461} C_DIS
LIN {X -0.008,Y -686.173,Z 1263.425,A 0.000,B 0.000,C 90.000,E1 112.408} C_DIS
LIN {X 0.205,Y -681.658,Z 1263.424,A 0.000,B 0.000,C 90.000,E1 112.280} C_DIS
LIN {X 0.297,Y -678.146,Z 1263.424,A 0.000,B 0.000,C 90.000,E1 112.206} C_DIS
LIN {X -0.189,Y -670.161,Z 1263.423,A 0.000,B 0.000,C 90.000,E1 112.206} C_DIS
LIN {X -0.238,Y -632.273,Z 1263.423,A 0.000,B 0.000,C 90.000,E1 112.206} C_DIS
LIN {X 0.081,Y -630.353,Z 1263.423,A 0.000,B 0.000,C 90.000,E1 112.099} C_DIS
LIN {X 0.272,Y -630.302,Z 1263.423,A 0.000,B 0.000,C 90.000,E1 112.078} C_DIS
LIN {X 0.222,Y -629.310,Z 1263.422,A 0.000,B 0.000,C 90.000,E1 111.972} C_DIS
LIN {X 0.178,Y -629.313,Z 1263.422,A 0.000,B 0.000,C 90.000,E1 111.972} C_DIS
LIN {X 0.100,Y -629.460,Z 1263.422,A 0.000,B 0.000,C 90.000,E1 111.844} C_DIS
LIN {X -0.002,Y -630.290,Z 1263.420,A 0.000,B 0.000,C 90.000,E1 111.663} C_DIS
LIN {X -0.184,Y -634.041,Z 1263.417,A 0.000,B 0.000,C 90.000,E1 111.046} C_DIS
LIN {X -0.179,Y -638.107,Z 1263.413,A 0.000,B 0.000,C 90.000,E1 110.429} C_DIS
LIN {X 0.299,Y -641.983,Z 1263.410,A 0.000,B 0.000,C 90.000,E1 109.758} C_DIS
LIN {X 0.021,Y -646.122,Z 1263.406,A 0.000,B 0.000,C 90.000,E1 109.033} C_DIS
LIN {X -0.218,Y -649.808,Z 1263.402,A 0.000,B 0.000,C 90.000,E1 108.308} C_DIS
LIN {X 0.266,Y -654.518,Z 1263.396,A 0.000,B 0.000,C 90.000,E1 107.275} C_DIS
LIN {X 0.095,Y -657.798,Z 1263.392,A 0.000,B 0.000,C 90.000,E1 106.551} C_DIS
LIN {X -0.128,Y -659.811,Z 1263.389,A 0.000,B 0.000,C 90.000,E1 106.079} C_DIS
LIN {X 0.206,Y -662.432,Z 1263.385,A 0.000,B 0.000,C 90.000,E1 105.315} C_DIS
LIN {X 0.192,Y -663.922,Z 1263.383,A 0.000,B 0.000,C 90.000,E1 104.828} C_DIS
LIN {X 0.014,Y -665.219,Z 1263.380,A 0.000,B 0.000,C 90.000,E1 104.356} C_DIS
LIN {X -0.238,Y -666.667,Z 1263.376,A 0.000,B 0.000,C 90.000,E1 103.647} C_DIS
LIN {X 0.250,Y -667.351,Z 1263.373,A 0.000,B 0.000,C 90.000,E1 103.119} C_DIS
LIN {X 0.094,Y -667.791,Z 1263.370,A 0.000,B 0.000,C 90.000,E1 102.647} C_DIS
LIN {X -0.060,Y -668.013,Z 1263.368,A 0.000,B 0.000,C 90.000,E1 102.175} C_DIS
LIN {X -0.352,Y -668.002,Z 1263.365,A 0.000,B 0.000,C 90.000,E1 101.715} C_DIS
LIN {X 0.070,Y -667.459,Z 1263.361,A 0.000,B 0.000,C 90.000,E1 100.950} C_DIS
LIN {X -0.215,Y -666.832,Z 1263.358,A 0.000,B 0.000,C 90.000,E1 100.489} C_DIS
LIN {X 0.275,Y -665.996,Z 1263.355,A 0.000,B 0.000,C 90.000,E1 99.962} C_DIS
LIN {X -0.014,Y -664.840,Z 1263.353,A 0.000,B 0.000,C 90.000,E1 99.500} C_DIS
LIN {X -0.199,Y -663.340,Z 1263.350,A 0.000,B 0.000,C 90.000,E1 99.029} C_DIS
LIN {X 0.256,Y -662.486,Z 1263.349,A 0.000,B 0.000,C 90.000,E1 98.746} C_DIS
LIN {X 0.050,Y -660.442,Z 1263.346,A 0.000,B 0.000,C 90.000,E1 98.276} C_DIS
LIN {X 0.282,Y -657.439,Z 1263.343,A 0.000,B 0.000,C 90.000,E1 97.644} C_DIS
LIN {X -0.052,Y -654.718,Z 1263.340,A 0.000,B 0.000,C 90.000,E1 97.182} C_DIS
LIN {X 0.245,Y -651.610,Z 1263.337,A 0.000,B 0.000,C 90.000,E1 96.663} C_DIS
LIN {X -0.236,Y -647.156,Z 1263.334,A 0.000,B 0.000,C 90.000,E1 96.087} C_DIS
LIN {X 0.010,Y -643.267,Z 1263.331,A 0.000,B 0.000,C 90.000,E1 95.568} C_DIS
LIN {X 0.102,Y -637.715,Z 1263.328,A 0.000,B 0.000,C 90.000,E1 94.935} C_DIS
LIN {X 0.312,Y -632.865,Z 1263.325,A 0.000,B 0.000,C 90.000,E1 94.416} C_DIS
LIN {X 0.020,Y -627.816,Z 1263.322,A 0.000,B 0.000,C 90.000,E1 93.955} C_DIS
LIN {X -0.144,Y -622.500,Z 1263.319,A 0.000,B 0.000,C 90.000,E1 93.498} C_DIS
LIN {X -0.077,Y -615.434,Z 1263.316,A 0.000,B 0.000,C 90.000,E1 92.922} C_DIS
LIN {X 0.234,Y -608.074,Z 1263.313,A 0.000,B 0.000,C 90.000,E1 92.350} C_DIS
LIN {X 0.179,Y -600.476,Z 1263.310,A 0.000,B 0.000,C 90.000,E1 91.835} C_DIS
LIN {X 0.084,Y -595.861,Z 1263.309,A 0.000,B 0.000,C 90.000,E1 91.547} C_DIS
LIN {X -0.252,Y -587.748,Z 1263.306,A 0.000,B 0.000,C 90.000,E1 91.146} C_DIS
LIN {X 0.173,Y -582.437,Z 1263.305,A 0.000,B 0.000,C 90.000,E1 90.859} C_DIS
LIN {X 0.211,Y -573.779,Z 1263.303,A 0.000,B 0.000,C 90.000,E1 90.516} C_DIS
LIN {X -0.198,Y -571.616,Z 1263.302,A 0.000,B 0.000,C 90.000,E1 90.458} C_DIS
LIN {X -0.226,Y -568.504,Z 1263.301,A 0.000,B 0.000,C 90.000,E1 90.172} C_DIS
LIN {X -0.264,Y -568.488,Z 1263.301,A 0.000,B 0.000,C 90.000,E1 90.172} C_DIS
LIN {X 0.190,Y -568.033,Z 1263.300,A 0.000,B 0.000,C 90.000,E1 89.885} C_DIS
LIN {X -0.071,Y -567.891,Z 1263.297,A 0.000,B 0.000,C 90.000,E1 89.484} C_DIS
LIN {X -0.151,Y -568.499,Z 1263.291,A 0.000,B 0.000,C 90.000,E1 88.396} C_DIS
LIN {X 0.195,Y -570.169,Z 1263.280,A 0.000,B 0.000,C 90.000,E1 86.445} C_DIS
LIN {X -0.111,Y -571.719,Z 1263.271,A 0.000,B 0.000,C 90.000,E1 84.837} C_DIS
LIN {X -0.074,Y -572.871,Z 1263.265,A 0.000,B 0.000,C 90.000,E1 83.742} C_DIS
LIN {X 0.173,Y -574.354,Z 1263.258,A 0.000,B 0.000,C 90.000,E1 82.356} C_DIS
LIN {X 0.078,Y -576.121,Z 1263.249,A 0.000,B 0.000,C 90.000,E1 80.735} C_DIS
LIN {X 0.251,Y -577.205,Z 1263.243,A 0.000,B 0.000,C 90.000,E1 79.634} C_DIS
LIN {X -0.024,Y -578.097,Z 1263.237,A 0.000,B 0.000,C 90.000,E1 78.578} C_DIS
LIN {X 0.162,Y -579.332,Z 1263.228,A 0.000,B 0.000,C 90.000,E1 76.937} C_DIS
LIN {X -0.055,Y -580.498,Z 1263.219,A 0.000,B 0.000,C 90.000,E1 75.338} C_DIS
LIN {X 0.048,Y -581.032,Z 1263.214,A 0.000,B 0.000,C 90.000,E1 74.519} C_DIS
LIN {X -0.034,Y -581.655,Z 1263.208,A 0.000,B 0.000,C 90.000,E1 73.449} C_DIS
LIN {X 0.116,Y -582.624,Z 1263.199,A 0.000,B 0.000,C 90.000,E1 71.819} C_DIS
LIN {X -0.258,Y -583.597,Z 1263.190,A 0.000,B 0.000,C 90.000,E1 70.242} C_DIS
LIN {X -0.350,Y -584.817,Z 1263.178,A 0.000,B 0.000,C 90.000,E1 68.103} C_DIS
LIN {X -0.211,Y -586.892,Z 1263.163,A 0.000,B 0.000,C 90.000,E1 65.409} C_DIS
LIN {X 0.276,Y -587.974,Z 1263.156,A 0.000,B 0.000,C 90.000,E1 64.024} C_DIS
LIN {X 0.188,Y -589.834,Z 1263.144,A 0.000,B 0.000,C 90.000,E1 61.897} C_DIS
LIN {X -0.169,Y -591.490,Z 1263.135,A 0.000,B 0.000,C 90.000,E1 60.333} C_DIS
LIN {X 0.000,Y -593.406,Z 1263.125,A 0.000,B 0.000,C 90.000,E1 58.456} C_DIS
LIN {X 0.318,Y -595.019,Z 1263.116,A 0.000,B 0.000,C 90.000,E1 56.834} C_DIS
LIN {X -0.063,Y -596.374,Z 1263.109,A 0.000,B 0.000,C 90.000,E1 55.548} C_DIS
LIN {X 0.253,Y -597.561,Z 1263.101,A 0.000,B 0.000,C 90.000,E1 54.196} C_DIS
LIN {X -0.242,Y -598.682,Z 1263.094,A 0.000,B 0.000,C 90.000,E1 52.924} C_DIS
LIN {X -0.361,Y -599.704,Z 1263.087,A 0.000,B 0.000,C 90.000,E1 51.618} C_DIS
LIN {X 0.137,Y -600.505,Z 1263.081,A 0.000,B 0.000,C 90.000,E1 50.517} C_DIS
LIN {X 0.158,Y -600.769,Z 1263.078,A 0.000,B 0.000,C 90.000,E1 49.989} C_DIS
LIN {X 0.183,Y -601.025,Z 1263.075,A 0.000,B 0.000,C 90.000,E1 49.461} C_DIS
LIN {X 0.025,Y -601.573,Z 1263.068,A 0.000,B 0.000,C 90.000,E1 48.162} C_DIS
LIN {X -0.128,Y -602.029,Z 1263.060,A 0.000,B 0.000,C 90.000,E1 46.863} C_DIS
LIN {X -0.096,Y -602.286,Z 1263.054,A 0.000,B 0.000,C 90.000,E1 45.810} C_DIS
LIN {X -0.056,Y -602.401,Z 1263.049,A 0.000,B 0.000,C 90.000,E1 44.757} C_DIS
LIN {X -0.016,Y -602.244,Z 1263.043,A 0.000,B 0.000,C 90.000,E1 43.704} C_DIS
LIN {X -0.396,Y -601.940,Z 1263.037,A 0.000,B 0.000,C 90.000,E1 42.690} C_DIS
LIN {X -0.142,Y -601.436,Z 1263.030,A 0.000,B 0.000,C 90.000,E1 41.353} C_DIS
LIN {X 0.155,Y -600.866,Z 1263.022,A 0.000,B 0.000,C 90.000,E1 40.011} C_DIS
LIN {X 0.068,Y -600.016,Z 1263.015,A 0.000,B 0.000,C 90.000,E1 38.705} C_DIS
LIN {X 0.098,Y -599.199,Z 1263.009,A 0.000,B 0.000,C 90.000,E1 37.649} C_DIS
LIN {X -0.260,Y -598.736,Z 1263.006,A 0.000,B 0.000,C 90.000,E1 37.156} C_DIS
LIN {X 0.093,Y -597.088,Z 1262.999,A 0.000,B 0.000,C 90.000,E1 35.804} C_DIS
LIN {X 0.183,Y -595.494,Z 1262.993,A 0.000,B 0.000,C 90.000,E1 34.739} C_DIS
LIN {X 0.295,Y -594.550,Z 1262.990,A 0.000,B 0.000,C 90.000,E1 34.199} C_DIS
LIN {X 0.013,Y -592.386,Z 1262.984,A 0.000,B 0.000,C 90.000,E1 33.166} C_DIS
LIN {X 0.313,Y -590.568,Z 1262.980,A 0.000,B 0.000,C 90.000,E1 32.339} C_DIS
LIN {X -0.339,Y -587.591,Z 1262.974,A 0.000,B 0.000,C 90.000,E1 31.337} C_DIS
LIN {X -0.100,Y -584.891,Z 1262.969,A 0.000,B 0.000,C 90.000,E1 30.512} C_DIS
LIN {X 0.153,Y -582.932,Z 1262.967,A 0.000,B 0.000,C 90.000,E1 29.951} C_DIS
LIN {X 0.181,Y -580.733,Z 1262.964,A 0.000,B 0.000,C 90.000,E1 29.411} C_DIS
LIN {X 0.119,Y -577.713,Z 1262.960,A 0.000,B 0.000,C 90.000,E1 28.743} C_DIS
LIN {X 0.372,Y -572.985,Z 1262.955,A 0.000,B 0.000,C 90.000,E1 27.769} C_DIS
LIN {X -0.036,Y -569.231,Z 1262.951,A 0.000,B 0.000,C 90.000,E1 27.129} C_DIS
LIN {X 0.038,Y -565.034,Z 1262.947,A 0.000,B 0.000,C 90.000,E1 26.437} C_DIS
LIN {X 0.123,Y -558.772,Z 1262.942,A 0.000,B 0.000,C 90.000,E1 25.463} C_DIS
LIN {X -0.004,Y -552.635,Z 1262.937,A 0.000,B 0.000,C 90.000,E1 24.643} C_DIS
LIN {X 0.161,Y -549.327,Z 1262.935,A 0.000,B 0.000,C 90.000,E1 24.207} C_DIS
LIN {X -0.067,Y -542.511,Z 1262.930,A 0.000,B 0.000,C 90.000,E1 23.387} C_DIS
LIN {X 0.266,Y -536.267,Z 1262.926,A 0.000,B 0.000,C 90.000,E1 22.642} C_DIS
LIN {X -0.015,Y -528.674,Z 1262.921,A 0.000,B 0.000,C 90.000,E1 21.844} C_DIS
LIN {X -0.012,Y -518.002,Z 1262.915,A 0.000,B 0.000,C 90.000,E1 20.737} C_DIS
LIN {X 0.122,Y -508.571,Z 1262.910,A 0.000,B 0.000,C 90.000,E1 19.758} C_DIS
LIN {X -0.197,Y -496.108,Z 1262.903,A 0.000,B 0.000,C 90.000,E1 18.598} C_DIS
LIN {X 0.015,Y -486.092,Z 1262.898,A 0.000,B 0.000,C 90.000,E1 17.638} C_DIS
LIN {X -0.112,Y -477.236,Z 1262.894,A 0.000,B 0.000,C 90.000,E1 16.858} C_DIS
LIN {X 0.115,Y -465.438,Z 1262.888,A 0.000,B 0.000,C 90.000,E1 15.788} C_DIS
LIN {X 0.196,Y -444.744,Z 1262.877,A 0.000,B 0.000,C 90.000,E1 13.883} C_DIS
LIN {X 0.095,Y -424.420,Z 1262.866,A 0.000,B 0.000,C 90.000,E1 11.883} C_DIS
LIN {X -0.141,Y -405.843,Z 1262.855,A 0.000,B 0.000,C 90.000,E1 9.905} C_DIS
LIN {X -0.171,Y -398.950,Z 1262.850,A 0.000,B 0.000,C 90.000,E1 9.095} C_DIS
LIN {X -0.110,Y -397.674,Z 1262.849,A 0.000,B 0.000,C 90.000,E1 8.916} C_DIS
LIN {X -0.068,Y -394.862,Z 1262.847,A 0.000,B 0.000,C 90.000,E1 8.454} C_DIS
LIN {X -0.094,Y -394.722,Z 1262.847,A 0.000,B 0.000,C 90.000,E1 8.398} C_DIS
LIN {X -0.132,Y -394.710,Z 1262.847,A 0.000,B 0.000,C 90.000,E1 8.398} C_DIS
LIN {X 0.180,Y -395.544,Z 1262.845,A 0.000,B 0.000,C 90.000,E1 8.106} C_DIS
LIN {X 0.129,Y -396.259,Z 1262.845,A 0.000,B 0.000,C 90.000,E1 7.992} C_DIS
LIN {X 0.098,Y -400.772,Z 1262.842,A 0.000,B 0.000,C 90.000,E1 7.587} C_DIS
LIN {X 0.147,Y -406.619,Z 1262.840,A 0.000,B 0.000,C 90.000,E1 7.182} C_DIS
LIN {X -0.008,Y -413.336,Z 1262.838,A 0.000,B 0.000,C 90.000,E1 6.777} C_DIS
LIN {X -0.127,Y -419.590,Z 1262.835,A 0.000,B 0.000,C 90.000,E1 6.372} C_DIS
LIN {X -0.130,Y -425.904,Z 1262.833,A 0.000,B 0.000,C 90.000,E1 5.910} C_DIS
LIN {X -0.051,Y -435.436,Z 1262.829,A 0.000,B 0.000,C 90.000,E1 5.163} C_DIS
LIN {X 0.193,Y -443.013,Z 1262.825,A 0.000,B 0.000,C 90.000,E1 4.531} C_DIS
LIN {X 0.037,Y -453.794,Z 1262.820,A 0.000,B 0.000,C 90.000,E1 3.669} C_DIS
LIN {X 0.066,Y -462.324,Z 1262.816,A 0.000,B 0.000,C 90.000,E1 2.922} C_DIS
LIN {X -0.035,Y -468.165,Z 1262.813,A 0.000,B 0.000,C 90.000,E1 2.407} C_DIS
LIN {X 0.115,Y -473.775,Z 1262.810,A 0.000,B 0.000,C 90.000,E1 1.835} C_DIS
LIN {X 0.031,Y -479.361,Z 1262.807,A 0.000,B 0.000,C 90.000,E1 1.260} C_DIS
LIN {X 0.092,Y -485.933,Z 1262.803,A 0.000,B 0.000,C 90.000,E1 0.516} C_DIS
LIN {X 0.000,Y -490.259,Z 1262.800,A 0.000,B 0.000,C 90.000,E1 360.000} C_DIS
LIN {X 0.029,Y -494.310,Z 1262.797,A 0.000,B 0.000,C 90.000,E1 359.484} C_DIS
LIN {X -0.078,Y -499.781,Z 1262.793,A 0.000,B 0.000,C 90.000,E1 358.740} C_DIS
LIN {X 0.074,Y -505.749,Z 1262.788,A 0.000,B 0.000,C 90.000,E1 357.822} C_DIS
LIN {X -0.138,Y -509.582,Z 1262.785,A 0.000,B 0.000,C 90.000,E1 357.249} C_DIS
LIN {X 0.129,Y -514.813,Z 1262.780,A 0.000,B 0.000,C 90.000,E1 356.331} C_DIS
LIN {X 0.011,Y -518.120,Z 1262.776,A 0.000,B 0.000,C 90.000,E1 355.755} C_DIS
LIN {X 0.147,Y -521.958,Z 1262.772,A 0.000,B 0.000,C 90.000,E1 355.008} C_DIS
LIN {X -0.203,Y -525.434,Z 1262.768,A 0.000,B 0.000,C 90.000,E1 354.318} C_DIS
LIN {X 0.016,Y -529.978,Z 1262.763,A 0.000,B 0.000,C 90.000,E1 353.280} C_DIS
LIN {X 0.038,Y -533.391,Z 1262.758,A 0.000,B 0.000,C 90.000,E1 352.413} C_DIS
LIN {X 0.098,Y -536.527,Z 1262.753,A 0.000,B 0.000,C 90.000,E1 351.546} C_DIS
LIN {X 0.188,Y -539.395,Z 1262.748,A 0.000,B 0.000,C 90.000,E1 350.679} C_DIS
LIN {X -0.134,Y -541.984,Z 1262.744,A 0.000,B 0.000,C 90.000,E1 349.859} C_DIS
LIN {X 0.006,Y -544.377,Z 1262.739,A 0.000,B 0.000,C 90.000,E1 348.993} C_DIS
LIN {X -0.169,Y -547.216,Z 1262.733,A 0.000,B 0.000,C 90.000,E1 347.881} C_DIS
LIN {X -0.075,Y -550.333,Z 1262.725,A 0.000,B 0.000,C 90.000,E1 346.464} C_DIS
LIN {X -0.283,Y -551.990,Z 1262.720,A 0.000,B 0.000,C 90.000,E1 345.644} C_DIS
LIN {X 0.196,Y -553.429,Z 1262.715,A 0.000,B 0.000,C 90.000,E1 344.755} C_DIS
LIN {X -0.259,Y -555.118,Z 1262.709,A 0.000,B 0.000,C 90.000,E1 343.685} C_DIS
LIN {X -0.001,Y -556.553,Z 1262.703,A 0.000,B 0.000,C 90.000,E1 342.543} C_DIS
LIN {X -0.249,Y -557.580,Z 1262.697,A 0.000,B 0.000,C 90.000,E1 341.456} C_DIS
LIN {X -0.071,Y -558.052,Z 1262.692,A 0.000,B 0.000,C 90.000,E1 340.604} C_DIS
LIN {X 0.114,Y -558.269,Z 1262.688,A 0.000,B 0.000,C 90.000,E1 339.752} C_DIS
LIN {X -0.223,Y -558.086,Z 1262.683,A 0.000,B 0.000,C 90.000,E1 338.954} C_DIS
LIN {X 0.176,Y -557.833,Z 1262.680,A 0.000,B 0.000,C 90.000,E1 338.358} C_DIS
LIN {X -0.177,Y -556.822,Z 1262.674,A 0.000,B 0.000,C 90.000,E1 337.283} C_DIS
LIN {X -0.315,Y -556.168,Z 1262.671,A 0.000,B 0.000,C 90.000,E1 336.741} C_DIS
LIN {X -0.173,Y -554.434,Z 1262.664,A 0.000,B 0.000,C 90.000,E1 335.613} C_DIS
LIN {X 0.178,Y -552.247,Z 1262.658,A 0.000,B 0.000,C 90.000,E1 334.460} C_DIS
LIN {X -0.007,Y -550.237,Z 1262.654,A 0.000,B 0.000,C 90.000,E1 333.640} C_DIS
LIN {X -0.238,Y -549.360,Z 1262.652,A 0.000,B 0.000,C 90.000,E1 333.384} C_DIS
LIN {X 0.033,Y -547.915,Z 1262.649,A 0.000,B 0.000,C 90.000,E1 332.794} C_DIS
LIN {X -0.205,Y -544.973,Z 1262.644,A 0.000,B 0.000,C 90.000,E1 331.975} C_DIS
LIN {X 0.285,Y -543.911,Z 1262.643,A 0.000,B 0.000,C 90.000,E1 331.641} C_DIS
LIN {X 0.253,Y -540.155,Z 1262.638,A 0.000,B 0.000,C 90.000,E1 330.795} C_DIS
LIN {X -0.155,Y -536.692,Z 1262.634,A 0.000,B 0.000,C 90.000,E1 330.127} C_DIS
LIN {X -0.125,Y -532.765,Z 1262.630,A 0.000,B 0.000,C 90.000,E1 329.410} C_DIS
LIN {X -0.171,Y -526.464,Z 1262.624,A 0.000,B 0.000,C 90.000,E1 328.408} C_DIS
LIN {X -0.016,Y -519.932,Z 1262.619,A 0.000,B 0.000,C 90.000,E1 327.375} C_DIS
LIN {X 0.127,Y -515.261,Z 1262.615,A 0.000,B 0.000,C 90.000,E1 326.628} C_DIS
LIN {X -0.076,Y -510.535,Z 1262.610,A 0.000,B 0.000,C 90.000,E1 325.801} C_DIS
LIN {X 0.070,Y -508.401,Z 1262.608,A 0.000,B 0.000,C 90.000,E1 325.341} C_DIS
LIN {X -0.022,Y -505.632,Z 1262.603,A 0.000,B 0.000,C 90.000,E1 324.609} C_DIS
LIN {X 0.023,Y -503.794,Z 1262.599,A 0.000,B 0.000,C 90.000,E1 323.863} C_DIS
LIN {X 0.105,Y -502.753,Z 1262.596,A 0.000,B 0.000,C 90.000,E1 323.256} C_DIS
LIN {X -0.118,Y -501.970,Z 1262.593,A 0.000,B 0.000,C 90.000,E1 322.683} C_DIS
LIN {X 0.121,Y -501.462,Z 1262.586,A 0.000,B 0.000,C 90.000,E1 321.457} C_DIS
LIN {X 0.080,Y -501.806,Z 1262.568,A 0.000,B 0.000,C 90.000,E1 318.162} C_DIS
LIN {X 0.088,Y -502.140,Z 1262.559,A 0.000,B 0.000,C 90.000,E1 316.662} C_DIS
LIN {X 0.038,Y -502.653,Z 1262.546,A 0.000,B 0.000,C 90.000,E1 314.271} C_DIS
LIN {X -0.154,Y -502.895,Z 1262.539,A 0.000,B 0.000,C 90.000,E1 313.095} C_DIS
LIN {X -0.250,Y -503.266,Z 1262.529,A 0.000,B 0.000,C 90.000,E1 311.310} C_DIS
LIN {X -0.176,Y -503.505,Z 1262.521,A 0.000,B 0.000,C 90.000,E1 309.806} C_DIS
LIN {X 0.160,Y -504.070,Z 1262.506,A 0.000,B 0.000,C 90.000,E1 307.076} C_DIS
LIN {X -0.087,Y -504.335,Z 1262.496,A 0.000,B 0.000,C 90.000,E1 305.311} C_DIS
LIN {X 0.195,Y -504.454,Z 1262.488,A 0.000,B 0.000,C 90.000,E1 303.785} C_DIS
LIN {X 0.088,Y -504.436,Z 1262.478,A 0.000,B 0.000,C 90.000,E1 302.005} C_DIS
LIN {X 0.142,Y -504.204,Z 1262.468,A 0.000,B 0.000,C 90.000,E1 300.207} C_DIS
LIN {X -0.124,Y -504.108,Z 1262.460,A 0.000,B 0.000,C 90.000,E1 298.743} C_DIS
LIN {X -0.125,Y -504.013,Z 1262.455,A 0.000,B 0.000,C 90.000,E1 297.847} C_DIS
LIN {X -0.198,Y -503.699,Z 1262.441,A 0.000,B 0.000,C 90.000,E1 295.463} C_DIS
LIN {X -0.126,Y -503.644,Z 1262.435,A 0.000,B 0.000,C 90.000,E1 294.259} C_DIS
LIN {X 0.119,Y -503.371,Z 1262.430,A 0.000,B 0.000,C 90.000,E1 293.334} C_DIS
LIN {X -0.097,Y -502.848,Z 1262.425,A 0.000,B 0.000,C 90.000,E1 292.461} C_DIS
LIN {X 0.225,Y -501.892,Z 1262.418,A 0.000,B 0.000,C 90.000,E1 291.227} C_DIS
LIN {X -0.017,Y -500.923,Z 1262.413,A 0.000,B 0.000,C 90.000,E1 290.355} C_DIS
LIN {X 0.091,Y -499.087,Z 1262.406,A 0.000,B 0.000,C 90.000,E1 289.141} C_DIS
LIN {X 0.055,Y -497.902,Z 1262.403,A 0.000,B 0.000,C 90.000,E1 288.544} C_DIS
LIN {X 0.068,Y -495.411,Z 1262.398,A 0.000,B 0.000,C 90.000,E1 287.638} C_DIS
LIN {X -0.108,Y -485.799,Z 1262.376,A 0.000,B 0.000,C 90.000,E1 283.703} C_DIS
LIN {X -0.170,Y -477.898,Z 1262.350,A 0.000,B 0.000,C 90.000,E1 279.086} C_DIS
LIN {X -0.011,Y -472.395,Z 1262.314,A 0.000,B 0.000,C 90.000,E1 272.522} C_DIS
LIN {X 0.082,Y -475.904,Z 1262.260,A 0.000,B 0.000,C 90.000,E1 262.818} C_DIS
LIN {X -0.060,Y -479.461,Z 1262.245,A 0.000,B 0.000,C 90.000,E1 260.038} C_DIS
LIN {X 0.117,Y -479.841,Z 1262.241,A 0.000,B 0.000,C 90.000,E1 259.398} C_DIS
LIN {X 0.152,Y -480.033,Z 1262.236,A 0.000,B 0.000,C 90.000,E1 258.465} C_DIS
LIN {X 0.144,Y -480.046,Z 1262.229,A 0.000,B 0.000,C 90.000,E1 257.229} C_DIS
LIN {X -0.156,Y -479.597,Z 1262.219,A 0.000,B 0.000,C 90.000,E1 255.408} C_DIS
LIN {X -0.048,Y -479.193,Z 1262.212,A 0.000,B 0.000,C 90.000,E1 254.157} C_DIS
LIN {X 0.052,Y -478.510,Z 1262.205,A 0.000,B 0.000,C 90.000,E1 252.906} C_DIS
LIN {X 0.054,Y -477.138,Z 1262.191,A 0.000,B 0.000,C 90.000,E1 250.423} C_DIS
LIN {X -0.206,Y -476.382,Z 1262.183,A 0.000,B 0.000,C 90.000,E1 248.901} C_DIS
LIN {X 0.101,Y -475.327,Z 1262.172,A 0.000,B 0.000,C 90.000,E1 246.997} C_DIS
LIN {X -0.282,Y -474.368,Z 1262.164,A 0.000,B 0.000,C 90.000,E1 245.485} C_DIS
LIN {X -0.045,Y -473.389,Z 1262.155,A 0.000,B 0.000,C 90.000,E1 243.896} C_DIS
LIN {X 0.037,Y -471.749,Z 1262.141,A 0.000,B 0.000,C 90.000,E1 241.385} C_DIS
LIN {X -0.228,Y -470.537,Z 1262.131,A 0.000,B 0.000,C 90.000,E1 239.537} C_DIS
LIN {X 0.202,Y -469.337,Z 1262.122,A 0.000,B 0.000,C 90.000,E1 237.916} C_DIS
LIN {X 0.289,Y -467.394,Z 1262.108,A 0.000,B 0.000,C 90.000,E1 235.388} C_DIS
LIN {X -0.194,Y -465.789,Z 1262.094,A 0.000,B 0.000,C 90.000,E1 232.924} C_DIS
LIN {X -0.127,Y -464.443,Z 1262.078,A 0.000,B 0.000,C 90.000,E1 230.070} C_DIS
LIN {X -0.063,Y -463.681,Z 1262.068,A 0.000,B 0.000,C 90.000,E1 228.162} C_DIS
LIN {X -0.265,Y -463.475,Z 1262.064,A 0.000,B 0.000,C 90.000,E1 227.553} C_DIS
LIN {X -0.252,Y -462.582,Z 1262.053,A 0.000,B 0.000,C 90.000,E1 225.648} C_DIS
LIN {X -0.010,Y -461.401,Z 1262.034,A 0.000,B 0.000,C 90.000,E1 222.123} C_DIS
LIN {X -0.020,Y -461.410,Z 1262.023,A 0.000,B 0.000,C 90.000,E1 220.216} C_DIS
LIN {X 0.172,Y -462.166,Z 1262.009,A 0.000,B 0.000,C 90.000,E1 217.649} C_DIS
LIN {X -0.090,Y -465.951,Z 1261.979,A 0.000,B 0.000,C 90.000,E1 212.291} C_DIS
LIN {X -0.003,Y -469.503,Z 1261.962,A 0.000,B 0.000,C 90.000,E1 209.127} C_DIS
LIN {X -0.062,Y -471.384,Z 1261.953,A 0.000,B 0.000,C 90.000,E1 207.564} C_DIS
LIN {X -0.250,Y -474.956,Z 1261.938,A 0.000,B 0.000,C 90.000,E1 204.771} C_DIS
LIN {X -0.058,Y -478.729,Z 1261.924,A 0.000,B 0.000,C 90.000,E1 202.259} C_DIS
LIN {X 0.157,Y -482.932,Z 1261.910,A 0.000,B 0.000,C 90.000,E1 199.758} C_DIS
LIN {X -0.110,Y -487.660,Z 1261.896,A 0.000,B 0.000,C 90.000,E1 197.330} C_DIS
LIN {X 0.006,Y -490.768,Z 1261.888,A 0.000,B 0.000,C 90.000,E1 195.788} C_DIS
LIN {X 0.018,Y -495.723,Z 1261.874,A 0.000,B 0.000,C 90.000,E1 193.355} C_DIS
LIN {X 0.173,Y -498.996,Z 1261.866,A 0.000,B 0.000,C 90.000,E1 191.827} C_DIS
LIN {X 0.153,Y -503.599,Z 1261.854,A 0.000,B 0.000,C 90.000,E1 189.726} C_DIS
LIN {X 0.141,Y -507.581,Z 1261.844,A 0.000,B 0.000,C 90.000,E1 187.936} C_DIS
LIN {X -0.127,Y -510.330,Z 1261.838,A 0.000,B 0.000,C 90.000,E1 186.777} C_DIS
LIN {X 0.049,Y -513.649,Z 1261.829,A 0.000,B 0.000,C 90.000,E1 185.277} C_DIS
LIN {X 0.236,Y -516.912,Z 1261.821,A 0.000,B 0.000,C 90.000,E1 183.784} C_DIS
LIN {X -0.061,Y -520.126,Z 1261.813,A 0.000,B 0.000,C 90.000,E1 182.350} C_DIS
LIN {X -0.255,Y -522.626,Z 1261.807,A 0.000,B 0.000,C 90.000,E1 181.203} C_DIS
LIN {X 0.027,Y -526.258,Z 1261.797,A 0.000,B 0.000,C 90.000,E1 179.427} C_DIS
LIN {X -0.102,Y -529.241,Z 1261.789,A 0.000,B 0.000,C 90.000,E1 177.993} C_DIS
LIN {X -0.168,Y -530.935,Z 1261.784,A 0.000,B 0.000,C 90.000,E1 177.135} C_DIS
LIN {X -0.209,Y -533.019,Z 1261.778,A 0.000,B 0.000,C 90.000,E1 175.988} C_DIS
LIN {X -0.144,Y -535.315,Z 1261.770,A 0.000,B 0.000,C 90.000,E1 174.546} C_DIS
LIN {X -0.073,Y -537.088,Z 1261.763,A 0.000,B 0.000,C 90.000,E1 173.394} C_DIS
LIN {X 0.078,Y -539.024,Z 1261.755,A 0.000,B 0.000,C 90.000,E1 171.951} C_DIS
LIN {X 0.267,Y -540.415,Z 1261.749,A 0.000,B 0.000,C 90.000,E1 170.792} C_DIS
LIN {X 0.016,Y -541.940,Z 1261.741,A 0.000,B 0.000,C 90.000,E1 169.398} C_DIS
LIN {X -0.109,Y -543.129,Z 1261.733,A 0.000,B 0.000,C 90.000,E1 167.993} C_DIS
LIN {X -0.005,Y -544.314,Z 1261.724,A 0.000,B 0.000,C 90.000,E1 166.284} C_DIS
LIN {X -0.054,Y -548.079,Z 1261.700,A 0.000,B 0.000,C 90.000,E1 162.054} C_DIS
LIN {X -0.151,Y -550.480,Z 1261.693,A 0.000,B 0.000,C 90.000,E1 160.659} C_DIS
LIN {X -0.202,Y -554.096,Z 1261.685,A 0.000,B 0.000,C 90.000,E1 159.263} C_DIS
LIN {X 0.227,Y -557.825,Z 1261.679,A 0.000,B 0.000,C 90.000,E1 158.103} C_DIS
LIN {X 0.202,Y -560.597,Z 1261.675,A 0.000,B 0.000,C 90.000,E1 157.411} C_DIS
LIN {X 0.210,Y -565.753,Z 1261.669,A 0.000,B 0.000,C 90.000,E1 156.305} C_DIS
LIN {X -0.086,Y -572.420,Z 1261.662,A 0.000,B 0.000,C 90.000,E1 155.101} C_DIS
LIN {X 0.105,Y -581.599,Z 1261.653,A 0.000,B 0.000,C 90.000,E1 153.589} C_DIS
LIN {X 0.019,Y -586.812,Z 1261.649,A 0.000,B 0.000,C 90.000,E1 152.794} C_DIS
LIN {X 0.038,Y -595.251,Z 1261.641,A 0.000,B 0.000,C 90.000,E1 151.463} C_DIS
LIN {X 0.060,Y -600.111,Z 1261.637,A 0.000,B 0.000,C 90.000,E1 150.667} C_DIS
LIN {X 0.205,Y -603.275,Z 1261.634,A 0.000,B 0.000,C 90.000,E1 150.127} C_DIS
LIN {X 0.263,Y -609.446,Z 1261.628,A 0.000,B 0.000,C 90.000,E1 149.076} C_DIS
LIN {X -0.338,Y -611.562,Z 1261.626,A 0.000,B 0.000,C 90.000,E1 148.742} C_DIS
LIN {X 0.010,Y -615.378,Z 1261.623,A 0.000,B 0.000,C 90.000,E1 148.074} C_DIS
LIN {X -0.270,Y -618.919,Z 1261.619,A 0.000,B 0.000,C 90.000,E1 147.454} C_DIS
LIN {X -0.205,Y -624.309,Z 1261.613,A 0.000,B 0.000,C 90.000,E1 146.421} C_DIS
LIN {X -0.062,Y -628.722,Z 1261.608,A 0.000,B 0.000,C 90.000,E1 145.515} C_DIS
LIN {X -0.231,Y -631.730,Z 1261.605,A 0.000,B 0.000,C 90.000,E1 144.895} C_DIS
LIN {X -0.008,Y -636.046,Z 1261.599,A 0.000,B 0.000,C 90.000,E1 143.863} C_DIS
LIN {X 0.244,Y -638.042,Z 1261.596,A 0.000,B 0.000,C 90.000,E1 143.336} C_DIS
LIN {X 0.031,Y -641.686,Z 1261.591,A 0.000,B 0.000,C 90.000,E1 142.351} C_DIS
LIN {X 0.253,Y -645.111,Z 1261.585,A 0.000,B 0.000,C 90.000,E1 141.331} C_DIS
LIN {X 0.019,Y -648.155,Z 1261.580,A 0.000,B 0.000,C 90.000,E1 140.356} C_DIS
LIN {X 0.260,Y -651.816,Z 1261.573,A 0.000,B 0.000,C 90.000,E1 139.094} C_DIS
LIN {X 0.063,Y -655.251,Z 1261.566,A 0.000,B 0.000,C 90.000,E1 137.877} C_DIS
LIN {X -0.086,Y -657.888,Z 1261.561,A 0.000,B 0.000,C 90.000,E1 136.905} C_DIS
LIN {X 0.229,Y -662.566,Z 1261.551,A 0.000,B 0.000,C 90.000,E1 135.162} C_DIS
LIN {X 0.177,Y -666.745,Z 1261.543,A 0.000,B 0.000,C 90.000,E1 133.704} C_DIS
LIN {X -0.264,Y -670.978,Z 1261.535,A 0.000,B 0.000,C 90.000,E1 132.285} C_DIS
LIN {X -0.150,Y -674.433,Z 1261.528,A 0.000,B 0.000,C 90.000,E1 131.067} C_DIS
LIN {X -0.390,Y -678.447,Z 1261.520,A 0.000,B 0.000,C 90.000,E1 129.644} C_DIS
LIN {X 0.368,Y -681.624,Z 1261.513,A 0.000,B 0.000,C 90.000,E1 128.382} C_DIS
LIN {X -0.202,Y -684.759,Z 1261.507,A 0.000,B 0.000,C 90.000,E1 127.237} C_DIS
LIN {X -0.348,Y -687.183,Z 1261.502,A 0.000,B 0.000,C 90.000,E1 126.297} C_DIS
LIN {X -0.276,Y -690.054,Z 1261.495,A 0.000,B 0.000,C 90.000,E1 125.105} C_DIS
LIN {X 0.199,Y -692.135,Z 1261.490,A 0.000,B 0.000,C 90.000,E1 124.119} C_DIS
LIN {X -0.392,Y -695.047,Z 1261.482,A 0.000,B 0.000,C 90.000,E1 122.752} C_DIS
LIN {X -0.240,Y -696.915,Z 1261.477,A 0.000,B 0.000,C 90.000,E1 121.799} C_DIS
LIN {X 0.185,Y -699.081,Z 1261.470,A 0.000,B 0.000,C 90.000,E1 120.590} C_DIS
LIN {X -0.049,Y -701.226,Z 1261.462,A 0.000,B 0.000,C 90.000,E1 119.205} C_DIS
LIN {X 0.090,Y -702.771,Z 1261.456,A 0.000,B 0.000,C 90.000,E1 118.025} C_DIS
LIN {X -0.017,Y -703.493,Z 1261.452,A 0.000,B 0.000,C 90.000,E1 117.334} C_DIS
LIN {X -0.075,Y -703.876,Z 1261.449,A 0.000,B 0.000,C 90.000,E1 116.873} C_DIS
LIN {X 0.148,Y -704.115,Z 1261.445,A 0.000,B 0.000,C 90.000,E1 116.155} C_DIS
LIN {X -0.223,Y -704.180,Z 1261.443,A 0.000,B 0.000,C 90.000,E1 115.720} C_DIS
LIN {X 0.347,Y -704.028,Z 1261.440,A 0.000,B 0.000,C 90.000,E1 115.207} C_DIS
LIN {X -0.020,Y -703.708,Z 1261.438,A 0.000,B 0.000,C 90.000,E1 114.771} C_DIS
LIN {X 0.263,Y -703.446,Z 1261.436,A 0.000,B 0.000,C 90.000,E1 114.515} C_DIS
LIN {X -0.105,Y -702.607,Z 1261.434,A 0.000,B 0.000,C 90.000,E1 114.079} C_DIS
LIN {X 0.168,Y -700.878,Z 1261.431,A 0.000,B 0.000,C 90.000,E1 113.590} C_DIS
LIN {X -0.202,Y -699.843,Z 1261.430,A 0.000,B 0.000,C 90.000,E1 113.387} C_DIS
LIN {X -0.068,Y -698.947,Z 1261.429,A 0.000,B 0.000,C 90.000,E1 113.259} C_DIS
LIN {X 0.180,Y -694.706,Z 1261.427,A 0.000,B 0.000,C 90.000,E1 112.770} C_DIS
LIN {X 0.306,Y -693.088,Z 1261.426,A 0.000,B 0.000,C 90.000,E1 112.642} C_DIS
LIN {X -0.270,Y -690.877,Z 1261.425,A 0.000,B 0.000,C 90.000,E1 112.589} C_DIS
LIN {X 0.058,Y -688.301,Z 1261.425,A 0.000,B 0.000,C 90.000,E1 112.461} C_DIS
LIN {X 0.174,Y -686.296,Z 1261.424,A 0.000,B 0.000,C 90.000,E1 112.386} C_DIS
LIN {X -0.149,Y -678.859,Z 1261.424,A 0.000,B 0.000,C 90.000,E1 112.259} C_DIS
LIN {X 0.257,Y -677.550,Z 1261.424,A 0.000,B 0.000,C 90.000,E1 112.206} C_DIS
LIN {X -0.063,Y -670.455,Z 1261.423,A 0.000,B 0.000,C 90.000,E1 112.206} C_DIS
LIN {X -0.108,Y -631.574,Z 1261.423,A 0.000,B 0.000,C 90.000,E1 112.206} C_DIS
LIN {X 0.125,Y -629.463,Z 1261.423,A 0.000,B 0.000,C 90.000,E1 112.099} C_DIS
LIN {X 0.079,Y -629.381,Z 1261.423,A 0.000,B 0.000,C 90.000,E1 112.099} C_DIS
LIN {X -0.096,Y -628.527,Z 1261.422,A 0.000,B 0.000,C 90.000,E1 112.025} C_DIS
LIN {X -0.140,Y -628.500,Z 1261.422,A 0.000,B 0.000,C 90.000,E1 112.025} C_DIS
LIN {X -0.211,Y -628.470,Z 1261.422,A 0.000,B 0.000,C 90.000,E1 111.897} C_DIS
LIN {X 0.104,Y -629.915,Z 1261.420,A 0.000,B 0.000,C 90.000,E1 111.535} C_DIS
LIN {X -0.015,Y -634.206,Z 1261.416,A 0.000,B 0.000,C 90.000,E1 110.844} C_DIS
LIN {X -0.188,Y -637.455,Z 1261.413,A 0.000,B 0.000,C 90.000,E1 110.355} C_DIS
LIN {X -0.155,Y -641.723,Z 1261.409,A 0.000,B 0.000,C 90.000,E1 109.631} C_DIS
LIN {X 0.354,Y -645.074,Z 1261.406,A 0.000,B 0.000,C 90.000,E1 108.960} C_DIS
LIN {X -0.072,Y -649.327,Z 1261.401,A 0.000,B 0.000,C 90.000,E1 108.127} C_DIS
LIN {X -0.220,Y -654.050,Z 1261.395,A 0.000,B 0.000,C 90.000,E1 107.149} C_DIS
LIN {X 0.043,Y -657.292,Z 1261.391,A 0.000,B 0.000,C 90.000,E1 106.386} C_DIS
LIN {X 0.003,Y -659.306,Z 1261.388,A 0.000,B 0.000,C 90.000,E1 105.898} C_DIS
LIN {X -0.307,Y -661.874,Z 1261.384,A 0.000,B 0.000,C 90.000,E1 105.190} C_DIS
LIN {X 0.054,Y -663.947,Z 1261.380,A 0.000,B 0.000,C 90.000,E1 104.426} C_DIS
LIN {X 0.040,Y -665.082,Z 1261.378,A 0.000,B 0.000,C 90.000,E1 103.939} C_DIS
LIN {X -0.131,Y -665.973,Z 1261.375,A 0.000,B 0.000,C 90.000,E1 103.467} C_DIS
LIN {X 0.202,Y -666.579,Z 1261.372,A 0.000,B 0.000,C 90.000,E1 102.952} C_DIS
LIN {X 0.044,Y -666.905,Z 1261.369,A 0.000,B 0.000,C 90.000,E1 102.479} C_DIS
LIN {X -0.113,Y -667.043,Z 1261.367,A 0.000,B 0.000,C 90.000,E1 102.007} C_DIS
LIN {X -0.273,Y -666.944,Z 1261.364,A 0.000,B 0.000,C 90.000,E1 101.535} C_DIS
LIN {X 0.218,Y -666.574,Z 1261.361,A 0.000,B 0.000,C 90.000,E1 101.007} C_DIS
LIN {X -0.074,Y -666.005,Z 1261.359,A 0.000,B 0.000,C 90.000,E1 100.546} C_DIS
LIN {X -0.246,Y -665.111,Z 1261.356,A 0.000,B 0.000,C 90.000,E1 100.074} C_DIS
LIN {X 0.114,Y -663.979,Z 1261.353,A 0.000,B 0.000,C 90.000,E1 99.557} C_DIS
LIN {X -0.182,Y -662.524,Z 1261.350,A 0.000,B 0.000,C 90.000,E1 99.095} C_DIS
LIN {X -0.280,Y -661.721,Z 1261.349,A 0.000,B 0.000,C 90.000,E1 98.859} C_DIS
LIN {X 0.066,Y -659.657,Z 1261.346,A 0.000,B 0.000,C 90.000,E1 98.341} C_DIS
